	// roll anticlockwise to reach limit
	7:
		IF NOT(m_jointMounted[4]) THEN  
			// set target joint position
			m_targetMountPos[4]:=curJntPos[4]+m_mountMotionAng;
			// check if reach limit 
			IF i_slaveArm.filtJntCurrent[4]>m_maxJntCurrent THEN 
				m_jointMounted[4]:=TRUE;
				m_jntLimitPos3 := curJntPos[4];
				m_targetMountPos[4]:=curJntPos[4];
				m_jntOTG[4].init(m_targetMountPos[4], 0,m_instruMountVel, m_instruMountAcc, g_slaveArmCtrlCycleTime);
			END_IF
		END_IF
		IF NOT(m_jointMounted[5]) THEN 
			// set target joint position
			m_targetMountPos[5]:=curJntPos[5]-m_mountMotionAng;
			// check if reach limit 
			IF i_slaveArm.filtJntCurrent[5]<- m_maxJntCurrent THEN 
				m_jointMounted[5]:=TRUE;
				m_jntLimitPos4 := curJntPos[5];
				m_targetMountPos[5]:=curJntPos[5];
				m_jntOTG[5].init(m_targetMountPos[5], 0,m_instruMountVel, m_instruMountAcc, g_slaveArmCtrlCycleTime);
			END_IF	
		END_IF
		
		// transit
		IF m_jointMounted[4] AND m_jointMounted[5] THEN
			m_yawJntCaliStatus := 8;
			m_jointMounted[4]:=FALSE;
			m_jointMounted[5]:= FALSE;
		END_IF
		
	8:// calculate center/calibarted position
		m_targetMountPos[4] := (m_jntLimitPos1 + m_jntLimitPos3)/2-i_slaveArm.instrument.instruTypeInfo.m_instruYawBacklash/2.0;
		m_targetMountPos[5] := (m_jntLimitPos2 + m_jntLimitPos4)/2+i_slaveArm.instrument.instruTypeInfo.m_instruYawBacklash/2.0;
		m_yawJntCaliStatus := 9;

	9:
		IF ABS(m_targetMountPos[4]-curJntPos[4]) <GVL_SlaveControlParameters.g_jntCtrlAngTolLow  AND
			ABS(m_targetMountPos[5]-curJntPos[5]) <GVL_SlaveControlParameters.g_jntCtrlAngTolLow  THEN
			m_targetMountPos[4] := curJntPos[4]+i_slaveArm.instrument.instruTypeInfo.m_instruYawBacklash;
			m_yawJntCaliStatus := 19;
		END_IF
	19:
		IF ABS(m_targetMountPos[4]-curJntPos[4]) <GVL_SlaveControlParameters.g_jntCtrlAngTolLow  AND
			ABS(m_targetMountPos[5]-curJntPos[5]) <GVL_SlaveControlParameters.g_jntCtrlAngTolLow  THEN
			m_yawJntCaliStatus := 20;
		END_IF
	20: 
		m_targetMountPos[4] := curJntPos[4]+22.50*g_deg2Rad;
		m_targetMountPos[5] := curJntPos[5]+22.50*g_deg2Rad;
		IF ABS(m_targetMountPos[4]-m_cmdJntPos[4]) <GVL_SlaveControlParameters.g_jntCtrlAngTolLow  AND
			ABS(m_targetMountPos[5]-m_cmdJntPos[5]) <GVL_SlaveControlParameters.g_jntCtrlAngTolLow  THEN
			m_targetMountPos[4]:=curJntPos[4];
			m_targetMountPos[5]:=curJntPos[5];
			m_jntOTG[1].init(m_targetMountPos[4], 0,m_instruMountVel, m_instruMountAcc, g_slaveArmCtrlCycleTime);
			m_jntOTG[2].init(m_targetMountPos[5], 0,m_instruMountVel, m_instruMountAcc, g_slaveArmCtrlCycleTime);
		m_yawJntCaliStatus := 21;
 		END_IF
	21:
		m_targetMountPos[4] := curJntPos[4]-0.35*i_slaveArm.instrument.instruTypeInfo.m_maxGripAngle-i_slaveArm.instrument.instruTypeInfo.m_instruYawBacklash-25*g_deg2Rad;
		m_targetMountPos[5] := curJntPos[5]-0.35*i_slaveArm.instrument.instruTypeInfo.m_maxGripAngle-i_slaveArm.instrument.instruTypeInfo.m_instruYawBacklash-25*g_deg2Rad;
		m_yawJntCaliStatus := 22;
    22:
		IF ABS(m_targetMountPos[4]-m_cmdJntPos[4]) <GVL_SlaveControlParameters.g_jntCtrlAngTolLow  AND
			ABS(m_targetMountPos[5]-m_cmdJntPos[5]) <GVL_SlaveControlParameters.g_jntCtrlAngTolLow  THEN
		m_yawJntCaliStatus := 23;
 		END_IF
	23:// calculate center/calibarted position
		m_targetMountPos[4] := (m_jntLimitPos1 + m_jntLimitPos3)/2-i_slaveArm.instrument.instruTypeInfo.m_instruYawBacklash/2.0;
		m_targetMountPos[5] := (m_jntLimitPos2 + m_jntLimitPos4)/2+i_slaveArm.instrument.instruTypeInfo.m_instruYawBacklash/2.0;
		m_yawJntCaliStatus := 24;

	24:
		IF ABS(m_targetMountPos[4]-curJntPos[4]) <GVL_SlaveControlParameters.g_jntCtrlAngTolLow  AND
			ABS(m_targetMountPos[5]-curJntPos[5]) <GVL_SlaveControlParameters.g_jntCtrlAngTolLow  THEN
			m_targetMountPos[4] := curJntPos[4]+i_slaveArm.instrument.instruTypeInfo.m_instruYawBacklash;
			m_yawJntCaliStatus := 25;
		END_IF
	25:
		IF ABS(m_targetMountPos[4]-curJntPos[4]) <GVL_SlaveControlParameters.g_jntCtrlAngTolLow  AND
			ABS(m_targetMountPos[5]-curJntPos[5]) <GVL_SlaveControlParameters.g_jntCtrlAngTolLow  THEN
			m_yawJntCaliStatus := 10;
		END_IF
		
	// close finger	
	10:
			m_targetMountPos[4] := curJntPos[4]+gripCloseAng;
			m_targetMountPos[5] := curJntPos[5]+gripCloseAng;
			m_yawJntCaliStatus := 11;
	11:
		IF ABS(m_targetMountPos[4]-curJntPos[4]) <GVL_SlaveControlParameters.g_jntCtrlAngTolLow  AND
			ABS(m_targetMountPos[5]-curJntPos[5]) <GVL_SlaveControlParameters.g_jntCtrlAngTolLow  THEN
			m_yawJntCaliStatus := -1;
		END_IF

END_CASE

// traj plan
m_jntOTG[4].run(m_targetMountPos[4],0.0, o_cmdAcc=>m_cmdJntAcc[4],o_cmdVel=>m_cmdJntVel[4],o_cmdPos=>m_cmdJntPos[4]);
m_jntOTG[5].run(m_targetMountPos[5],0.0, o_cmdAcc=>m_cmdJntAcc[5],o_cmdVel=>m_cmdJntVel[5],o_cmdPos=>m_cmdJntPos[5]);
END_METHOD

END_FUNCTION_BLOCK

// ---- FBs_SlaveControllers/FB_SlaveArmCtrlBase.TcPOU
// Slave Arm Base Controller, Hold at Current Posture
FUNCTION_BLOCK FB_SlaveArmCtrlBase IMPLEMENTS I_SlaveArmCtrl
VAR_INPUT
END_VAR
VAR_OUTPUT
END_VAR
VAR
	// flag if the controller has finished all its jobs
	m_isFinished:BOOL:=FALSE;
	
	// controller execute time period
	m_timePeriod :LREAL:=0;
	
	// flag to hold last commands
	m_holdLastCmds :BOOL := FALSE;
	
	// arm control data
	// NOTE: simulated joint position is usd for kinematic controller 
	//		while command joint position is used for real robot controller
	// 		They are identical for the most time, but in some cases, simulated position is filted to get command one 
	m_simJntPos :Vec8d; 
	m_cmdJntPos : VEC8d; 
	m_cmdJntVel : VEC8d;
	m_cmdJntAcc : VEC8d;
	m_cmdJntTrq : VEC8d;
	m_jntOPMode : Vec8i;
	m_jntEnableFlag :Vec8i;
	m_cmdCartPose : ST_Frame;
	m_cmdCartTwist : Vec6d;
	m_FFJntTrq :Vec8d;
	
END_VAR

// override this function in each exact controller
METHOD PROTECTED calcCmdJntPos : BOOL
VAR_IN_OUT CONSTANT
	// endoscope pose in cart coordinate
	i_endoscopePose : ST_Frame;
	
	// master arm data
	i_masterStatus :ST_MasterStatus;
	
	// setup arm data
	i_setupStatus: ST_SetupStatus;
	
	// slave arm data
	i_slaveArm :FB_SlaveArm;
END_VAR
IF isFinished THEN
	RETURN;
END_IF
END_METHOD

// override this function in each exact controller
METHOD PROTECTED calcCmdJntTrq : BOOL
VAR_IN_OUT CONSTANT
	// endoscope pose in cart coordinate
	i_endoscopePose : ST_Frame;
	
	// master arm data
	i_masterStatus :ST_MasterStatus;
	
	// setup arm data
	i_setupStatus: ST_SetupStatus;
	
	// slave arm data
	i_slaveArm :FB_SlaveArm;
END_VAR
IF isFinished THEN
	RETURN;
END_IF

// set joint torque to zero in default
m_cmdJntTrq := g_zeroVec8d;
END_METHOD

METHOD checkToHoldLastCmds : BOOL
VAR_IN_OUT CONSTANT
	i_slaveArm :FB_SlaveArm;
END_VAR
VAR
	j:INT;
	maxJntErr:LREAL;
	jntCtrlErr:Vec8d;
END_VAR
// check if to hold the command joint position unchanged
vecSub(i_slaveArm.m_cmdJntPos, i_slaveArm.m_curJntPos,jntCtrlErr);
maxJntErr:=0.0;
FOR j:=1 TO g_sJntNum DO
	maxJntErr:= MAX(maxJntErr, ABS(jntCtrlErr[j]));
END_FOR

checkToHoldLastCmds := (maxJntErr<GVL_SlaveControlParameters.g_jntCtrlErrForCmdHold);
END_METHOD

METHOD copyCmds : BOOL
VAR_IN_OUT 
	r_slaveArmCtrlCmd :ST_SlaveArmCtrlCmds;
END_VAR
r_slaveArmCtrlCmd.m_jntEnableFlag :=m_jntEnableFlag;
r_slaveArmCtrlCmd.m_cmdCartPose:=m_cmdCartPose;
r_slaveArmCtrlCmd.m_cmdCartTwist:=m_cmdCartTwist;
r_slaveArmCtrlCmd.m_simJntPos:=m_simJntPos;
r_slaveArmCtrlCmd.m_cmdJntPos:=m_cmdJntPos;
r_slaveArmCtrlCmd.m_cmdJntVel:=m_cmdJntVel;
r_slaveArmCtrlCmd.m_cmdJntAcc:=m_cmdJntAcc;
r_slaveArmCtrlCmd.m_cmdJntTrq:=m_cmdJntTrq;
r_slaveArmCtrlCmd.m_jntOPMode:=m_jntOPMode;
r_slaveArmCtrlCmd.m_FFJntTrq:=m_FFJntTrq;
END_METHOD

// call this function to add friction compensation to m_cmdJntTrq
METHOD enableFrictionCompensation : BOOL
VAR_IN_OUT CONSTANT
	i_slaveArm :FB_SlaveArm;
END_VAR

VAR
	i:INT;
	frictionScale :LREAL;
END_VAR
// add joint friction compensation
FOR i:=1 TO g_sJntNum DO
	frictionScale :=LIMIT(-1.0, i_slaveArm.curJntVel[i]/g_fullFrictionVel,1.0);
	m_cmdJntTrq[i]:=m_cmdJntTrq[i]+frictionScale * g_frictionCompScale * GVL_SlaveArmDynamics.g_slaveJntFriction[i_slaveArm.armIdx, i];
END_FOR
END_METHOD

// override this function in each exact controller
// NOTICE: set joint control mode here, and do some initialization if needed
METHOD PUBLIC init : BOOL
VAR_IN_OUT CONSTANT
	i_slaveArm	:FB_SlaveArm;
END_VAR
VAR_IN_OUT 
	r_slaveArmCtrlCmd :ST_SlaveArmCtrlCmds;
END_VAR
m_timePeriod:=0;
m_jntEnableFlag :=g_onesVec8i;
m_jntEnableFlag[1] := 0;
m_jntEnableFlag[2] := 0;
m_jntEnableFlag[3] := 0;
m_jntOPMode:=g_slaveAllPosMode;
m_cmdCartPose:=i_slaveArm.curCartPose;
m_cmdCartTwist:=g_zeroVec6d;
IF FALSE = m_holdLastCmds THEN
	m_cmdJntPos:=i_slaveArm.curJntPos;
ELSE
	m_cmdJntPos:=r_slaveArmCtrlCmd.m_cmdJntPos;
END_IF
m_simJntPos := m_cmdJntPos;
m_cmdJntVel:=g_zeroVec8d;
m_cmdJntAcc:=g_zeroVec8d;
m_cmdJntTrq:=g_zeroVec8d;
m_FFJntTrq :=g_zeroVec8d;

// update commands to arm
copyCmds(r_slaveArmCtrlCmd);
END_METHOD

PROPERTY isFinished : BOOL
GET
isFinished:=m_isFinished;
END_GET
END_PROPERTY

{warning '添加方法实现'}
METHOD reset : BOOL
m_isFinished:=FALSE;
m_timePeriod:=0;
END_METHOD

{warning '添加方法实现'}
METHOD run : BOOL
VAR_IN_OUT CONSTANT
	i_endoscopePose : ST_Frame;
	i_masterStatus :ST_MasterStatus;
	i_setupStatus: ST_SetupStatus;
	i_slaveArm :FB_SlaveArm;
END_VAR
VAR_IN_OUT
	r_slaveArmCtrlCmd :ST_SlaveArmCtrlCmds;
END_VAR
VAR
	i:INT;
END_VAR
IF m_isFinished THEN
	RETURN;
END_IF

// check if arm enabled
IF FALSE = i_slaveArm.isEnabled(m_jntEnableFlag) THEN
	RETURN;
END_IF

// calculate command joint position--Motion control
calcCmdJntPos(i_endoscopePose, i_masterStatus, i_setupStatus, i_slaveArm);

// calculate command joint torque -- Force control
calcCmdJntTrq(i_endoscopePose, i_masterStatus, i_setupStatus, i_slaveArm);

// update commands to arm
copyCmds(r_slaveArmCtrlCmd);

// update time period
m_timePeriod := m_timePeriod+g_slaveArmCtrlCycleTime;
END_METHOD

PROPERTY timePeriod : Lreal
GET
timePeriod := m_timePeriod;
END_GET
END_PROPERTY

END_FUNCTION_BLOCK

// ---- FBs_SlaveControllers/FB_SlaveCtrlInstruEndoscopeTest.TcPOU
// Brief: Slave Arm test
FUNCTION_BLOCK PUBLIC FB_SlaveCtrlInstruEndoscopeTest EXTENDS FB_SlaveArmCtrlBase
VAR
																
	// final target DH joint position and grip angle
	m_targetDHJntPos:Vec3d;
	m_targetGripAng:LREAL;
	m_targetGripForceLevel :LREAL :=0;
	m_maxGripCurrent:LREAL:=350.0;
	m_maxGripCtrlCurrent:LREAL:=540.0;
	
	// interploated command joint position and grip angle 
	m_cmdDHJntPos :Vec6d;
	m_cmdDHJntVel :Vec6d;
	m_cmdGripAng:LREAL;

	// last joint position 
	m_lastCmdJntPos :Vec8d ;
	
	// instrument controller
	m_instruController : FB_BasicInstruControl;
	m_usKnifeController : FB_UltrosonicKnifeControl;
	m_instruCmdJntPos,m_instruCmdJntVel : Vec5d;
	m_instruCmdJntTrq :Vec5d;
	
	// OTG
	m_DHJntOTG:ARRAY[1..3] OF FB_secOrdTrajFilter;
	m_gripAngleOTG : FB_secOrdTrajFilter;
	m_maxJntVel:Vec3d:=[3(2.0)];
	m_maxJntAcc:Vec3d:=[3(4.0)];
	
	// instrument tyep
	m_instruType : E_InstrumentType;

	
	m_endoscopeAdjustment:BOOL;
	m_endoscopeOverturn:BOOL;
	m_endoscopeAdjustmentLast:BOOL;
	m_endoscopeOverturnLast:BOOL;
	
	m_tonEndoscopeOverturn:TON;
	m_endoscopeOverturn30:BOOL;
	m_endoscopeOverturn30Last:BOOL;
END_VAR

METHOD PROTECTED calcCmdJntPos : BOOL
VAR_IN_OUT CONSTANT
	i_endoscopePose : ST_Frame;
	i_masterStatus :ST_MasterStatus;
	i_setupStatus: ST_SetupStatus;
	i_slaveArm :FB_SlaveArm;
END_VAR

VAR 
	i:INT :=0;

END_VAR
//0/30°调整信号
IF (i_slaveArm.m_panelInstrumentOnIO  = 111) THEN      
	m_endoscopeAdjustment:=TRUE;
ELSE
	m_endoscopeAdjustment:=FALSE;
END_IF
//内窥镜翻转调整信号
IF (i_slaveArm.m_panelInstrumentOnIO =95) THEN    
	m_endoscopeOverturn:=TRUE;
ELSE
	m_endoscopeOverturn:=FALSE;
END_IF
m_tonEndoscopeOverturn(IN:=i_slaveArm.m_panelInstrumentOnIO  = 111,PT:=T#3S);
IF m_tonEndoscopeOverturn.Q THEN
	m_endoscopeOverturn30:=TRUE;
ELSE
	m_endoscopeOverturn30:=FALSE;
END_IF
//0/30°镜切换
IF m_endoscopeAdjustment AND NOT m_endoscopeAdjustmentLast THEN
	IF GVL_InstruTestUIVars.g_endoscopeAngle=0 THEN
		GVL_InstruTestUIVars.g_endoscopeAngle:=30;
	ELSE
		GVL_InstruTestUIVars.g_endoscopeAngle:=0;
	END_IF
END_IF
IF m_endoscopeOverturn30 AND NOT m_endoscopeOverturn30Last THEN
	IF GVL_InstruTestUIVars.g_endoscopeUpturn30FlagBit THEN
		m_targetDHJntPos[1]:=i_slaveArm.curDHJntPos[4]+30*g_deg2rad;
		GVL_InstruTestUIVars.g_endoscopeUpturn30FlagBit:=0;
	ELSE
		m_targetDHJntPos[1]:=i_slaveArm.curDHJntPos[4]-30*g_deg2rad;	
		GVL_InstruTestUIVars.g_endoscopeUpturn30FlagBit:=1;
	END_IF
END_IF
//内窥镜翻转信号
IF m_endoscopeOverturn AND NOT m_endoscopeOverturnLast THEN
	IF GVL_InstruTestUIVars.g_endoscopeUpturnFlagBit THEN
		m_targetDHJntPos[1]:=i_slaveArm.curDHJntPos[4]+180*g_deg2rad;
		GVL_InstruTestUIVars.g_endoscopeUpturnFlagBit:=0;
	ELSE
		m_targetDHJntPos[1]:=i_slaveArm.curDHJntPos[4]-180*g_deg2rad;	
		GVL_InstruTestUIVars.g_endoscopeUpturnFlagBit:=1;
	END_IF
END_IF
IF GVL_InstruTestUIVars.g_startEndoscopeTest THEN 
	m_targetDHJntPos[1]:=i_slaveArm.curDHJntPos[4]+GVL_InstruTestUIVars.g_cycleEndoscopeTest*2*pi;
	GVL_InstruTestUIVars.g_startEndoscopeTest:=0;
END_IF
m_endoscopeOverturnLast:=m_endoscopeOverturn;
m_endoscopeAdjustmentLast:=m_endoscopeAdjustment;
m_endoscopeOverturn30Last:=m_endoscopeOverturn30;
// run OTG
FOR i:=1 TO 3  DO
	m_DHJntOTG[i].run(m_targetDHJntPos[i],0.0, o_cmdAcc=>,o_cmdVel=>m_cmdDHJntVel[i],o_cmdPos=> m_cmdDHJntPos[i+3]);
END_FOR
m_gripAngleOTG.run(m_targetGripAng,0.0, o_cmdAcc=>,o_cmdVel=>,o_cmdPos=>m_cmdGripAng);
// calculate target motor joint position from DH joint position
i_slaveArm.instrument.instruIK(m_cmdDHJntPos,m_cmdGripAng, o_jntPos=>m_cmdJntPos);

// command velocity
vecSub(m_cmdJntPos, m_lastCmdJntPos, m_cmdJntVel);
vecSelfMultiNum(m_cmdJntVel, g_slaveArmCtrlFreq);
m_lastCmdJntPos:=m_cmdJntPos;
END_METHOD

// override this function in each exact controller
METHOD PROTECTED calcCmdJntTrq : BOOL
VAR_IN_OUT CONSTANT
	i_endoscopePose : ST_Frame;
	i_masterStatus :ST_MasterStatus;
	i_setupStatus: ST_SetupStatus;
	i_slaveArm :FB_SlaveArm;
END_VAR

VAR 
	nullspaceMat :Mat7d;
	ctrlTrq : Vec7d;
	i : int ;
END_VAR
// set joint torque to zero in default
m_cmdJntTrq := g_zeroVec8d;

// instrument joint control
FOR i:=1 TO 5 DO 
	m_instruCmdJntPos[i]:=m_cmdJntPos[i+3];
	m_instruCmdJntVel[i]:=m_cmdJntVel[i+3];
END_FOR

IF i_slaveArm.instrument.instruType = InstruType_UltrasoundKnifeS OR i_slaveArm.instrument.instruType = InstruType_UltrasoundKnifeU THEN
	m_usKnifeController.run(m_instruCmdJntPos,m_instruCmdJntVel, m_targetGripForceLevel, i_slaveArm, o_cmdJntTrq=>m_instruCmdJntTrq);
ELSE
	m_instruController.run(m_instruCmdJntPos,m_instruCmdJntVel, m_cmdDHJntPos[6], m_cmdDHJntVel[6], m_targetGripForceLevel, i_slaveArm, o_cmdJntTrq=>m_instruCmdJntTrq);
END_IF

FOR i:=1 TO 5 DO
	m_cmdJntTrq[i+3]:=m_instruCmdJntTrq[i];
	m_cmdJntTrq[6]:=0;
END_FOR
END_METHOD

METHOD PUBLIC init : BOOL
VAR_IN_OUT CONSTANT
	i_slaveArm	:FB_SlaveArm;
END_VAR
VAR_IN_OUT 
	r_slaveArmCtrlCmd :ST_SlaveArmCtrlCmds;
END_VAR

VAR
	i:int;
END_VAR
SUPER^.Init(i_slaveArm,r_slaveArmCtrlCmd);
m_lastCmdJntPos:=m_cmdJntPos;
m_jntOPMode[1] := DriverOPMode_PosTrq;
m_jntOPMode[2] := DriverOPMode_PosTrq;
m_jntOPMode[3] := DriverOPMode_PosTrq;
m_jntOPMode[4] := DriverOPMode_Trq;
m_jntOPMode[5] := DriverOPMode_Trq;
m_jntOPMode[6] := DriverOPMode_Trq;
m_jntOPMode[7] := DriverOPMode_Trq;
m_jntOPMode[8] := DriverOPMode_Trq;

m_cmdDHJntPos :=i_slaveArm.curDHJntPos;
m_cmdDHJntVel :=g_zeroVec6d;
m_targetGripAng := i_slaveArm.curGripAngle;
m_targetDHJntPos[1] := i_slaveArm.curDHJntPos[4];
m_targetDHJntPos[2] := i_slaveArm.curDHJntPos[5];
m_targetDHJntPos[3] := i_slaveArm.curDHJntPos[6];

// init instrument controller
m_instruController.init(i_slaveArm,m_maxGripCurrent,m_maxGripCtrlCurrent);
m_usKnifeController.init(i_slaveArm);

FOR i:=1 TO 3  DO
	m_DHJntOTG[i].init(m_cmdDHJntPos[i+3], 0, m_maxJntVel[i], m_maxJntAcc[i], g_slaveArmCtrlCycleTime);
END_FOR

m_gripAngleOTG.init(m_targetGripAng, 0, 2*m_maxJntVel[3], 2*m_maxJntAcc[3], g_slaveArmCtrlCycleTime);
// update commands to arm
copyCmds(r_slaveArmCtrlCmd);
END_METHOD

PROPERTY InstruBacklash : Vec5d
GET
IF m_instruType = InstruType_UltrasoundKnifeS OR m_instruType = InstruType_UltrasoundKnifeU THEN
	instruBacklash := g_zeroVec5d;
ELSE
	instruBacklash := m_instruController.m_jntBacklash;
END_IF
END_GET
END_PROPERTY

END_FUNCTION_BLOCK

// ---- FBs_SlaveControllers/FB_SlaveCtrlInstruManualTest.TcPOU
// Brief: Slave Arm test
FUNCTION_BLOCK PUBLIC FB_SlaveCtrlInstruManualTest EXTENDS FB_SlaveArmCtrlBase
VAR
																
	// final target DH joint position and grip angle
	m_targetDHJntPos:Vec3d;
	m_targetGripAng:LREAL;
	m_targetGripForceLevel :LREAL :=0;
	
	// interploated command joint position and grip angle 
	m_cmdDHJntPos :Vec6d;
	m_cmdDHJntVel :Vec6d;
	m_cmdGripAng:LREAL;

	// last joint position 
	m_lastCmdJntPos :Vec8d ;
	
	// instrument controller
	m_instruController : FB_BasicInstruControl;
	m_usKnifeController : FB_UltrosonicKnifeControl;
	m_instruCmdJntPos,m_instruCmdJntVel : Vec5d;
	m_instruCmdJntTrq :Vec5d;
	
	// OTG
	m_DHJntOTG:ARRAY[1..3] OF FB_secOrdTrajFilter;
	m_gripAngleOTG : FB_secOrdTrajFilter;
	m_maxJntVel:Vec3d:=[3(2.0)];
	m_maxJntAcc:Vec3d:=[3(4.0)];
	
	// instrument tyep
	m_instruType : E_InstrumentType;
	bStart: BOOL;
	iStep: INT;
	fbTon: TON;

	m_maxGripCurrent:LREAL:=350.0;
	m_maxGripCtrlCurrent:LREAL:=540.0;
END_VAR

METHOD PROTECTED calcCmdJntPos : BOOL
VAR_IN_OUT CONSTANT
	i_endoscopePose : ST_Frame;
	i_masterStatus :ST_MasterStatus;
	i_setupStatus: ST_SetupStatus;
	i_slaveArm :FB_SlaveArm;
END_VAR

VAR 
	i:INT :=0;
	errThres :LREAL;
	m_targetDHJntPosLast: Vec3d;
	m_curCmdDHJntPos: Vec3d;
	m_compensationAngleDH: Vec3d;
	m_targetGripAngLast: LREAL;
	m_curCmdAng: LREAL;

END_VAR
// determine target DH joint position and gripper motion
IF GVL_InstruTestUIVars.g_moveToSetPosFlag THEN
	m_targetDHJntPos[1] := GVL_InstruTestUIVars.g_targetRollAng*g_deg2rad;
	m_targetDHJntPos[2] := (GVL_InstruTestUIVars.g_targetPitchAng-90)*g_deg2rad;
	m_targetDHJntPos[3] := GVL_InstruTestUIVars.g_targetYawAng*g_deg2rad;
	IF GVL_InstruTestUIVars.g_targetGripAng>-15 AND GVL_InstruTestUIVars.g_targetGripAng<100  THEN 
		m_targetGripAng := GVL_InstruTestUIVars.g_targetGripAng*g_deg2rad;
		m_targetGripForceLevel:=0;
	ELSIF GVL_InstruTestUIVars.g_targetGripAng<=-15 AND GVL_InstruTestUIVars.g_targetGripAng>=-100 THEN 
		m_targetGripAng := -15*g_deg2rad;
		m_targetGripForceLevel := LIMIT(0, ABS(GVL_InstruTestUIVars.g_targetGripAng), 100);
	ELSIF GVL_InstruTestUIVars.g_targetGripAng<-101 THEN 
		m_targetGripAng := 60 *g_deg2rad;
		m_targetGripForceLevel := LIMIT(-100, 100+GVL_InstruTestUIVars.g_targetGripAng, 0);
	END_IF
ELSIF GVL_InstruTestUIVars.g_gripperOpenFlag THEN
	m_targetGripAng := i_slaveArm.instrument.instruTypeInfo.m_maxGripAngle;
	m_targetGripForceLevel :=0;
ELSIF GVL_InstruTestUIVars.g_gripperCloseFlag THEN
	m_targetGripAng := 0;
	m_targetGripForceLevel :=0;
ELSIF GVL_InstruTestUIVars.g_maxGripForceFlag THEN
	m_targetGripAng := -45*g_deg2rad;
	m_targetGripForceLevel :=100;
END_IF

IF GVL_InstruTestUIVars.m_cycleStart THEN 
	bStart:=TRUE;
	GVL_InstruTestUIVars.m_cycleStart:=FALSE;
END_IF
IF GVL_InstruTestUIVars.m_cycleStop THEN 
	bStart:=FALSE;
	GVL_InstruTestUIVars.m_cycleStop:=FALSE;
END_IF
fbTon(IN:=iStep=10,PT:=T#1S);
IF bStart THEN
	CASE iStep OF 
		0:
			m_targetGripAng := i_slaveArm.instrument.instruTypeInfo.m_maxGripAngle;
			m_targetGripForceLevel :=0;
			iStep:=5;
		5:
		    IF ABS(m_cmdGripAng- m_targetGripAng)< g_jntCtrlAngTolLow THEN
				iStep:=10;
			END_IF
		10:
			IF fbTon.Q THEN
				m_targetGripAng := -90*g_deg2rad;
				m_targetGripForceLevel :=0;
				iStep:=15;
			END_IF
		15:
		    IF ABS(m_cmdGripAng- m_targetGripAng)< g_jntCtrlAngTolLow THEN
				iStep:=0;
			END_IF
	END_CASE
END_IF
// run OTG
FOR i:=1 TO 3  DO
	m_DHJntOTG[i].run(m_targetDHJntPos[i],0.0, o_cmdAcc=>,o_cmdVel=>m_cmdDHJntVel[i],o_cmdPos=> m_cmdDHJntPos[i+3]);
END_FOR
m_gripAngleOTG.run(m_targetGripAng,0.0, o_cmdAcc=>,o_cmdVel=>,o_cmdPos=>m_cmdGripAng);

// calculate target motor joint position from DH joint position
i_slaveArm.instrument.instruIK(m_cmdDHJntPos,m_cmdGripAng, o_jntPos=>m_cmdJntPos);

// command velocity
vecSub(m_cmdJntPos, m_lastCmdJntPos, m_cmdJntVel);
vecSelfMultiNum(m_cmdJntVel, g_slaveArmCtrlFreq);
m_lastCmdJntPos:=m_cmdJntPos;
END_METHOD

// override this function in each exact controller
METHOD PROTECTED calcCmdJntTrq : BOOL
VAR_IN_OUT CONSTANT
	i_endoscopePose : ST_Frame;
	i_masterStatus :ST_MasterStatus;
	i_setupStatus: ST_SetupStatus;
	i_slaveArm :FB_SlaveArm;
END_VAR

VAR 
	nullspaceMat :Mat7d;
	ctrlTrq : Vec7d;
	i : int ;
END_VAR
// set joint torque to zero in default
m_cmdJntTrq := g_zeroVec8d;

// instrument joint control
FOR i:=1 TO 5 DO 
	m_instruCmdJntPos[i]:=m_cmdJntPos[i+3];
	m_instruCmdJntVel[i]:=m_cmdJntVel[i+3];
END_FOR

IF i_slaveArm.instrument.instruType = InstruType_UltrasoundKnifeS OR i_slaveArm.instrument.instruType = InstruType_UltrasoundKnifeU THEN
	m_usKnifeController.run(m_instruCmdJntPos,m_instruCmdJntVel, m_targetGripForceLevel, i_slaveArm, o_cmdJntTrq=>m_instruCmdJntTrq);
ELSE
	m_instruController.run(m_instruCmdJntPos,m_instruCmdJntVel, m_cmdDHJntPos[6], m_cmdDHJntVel[6], m_targetGripForceLevel, i_slaveArm, o_cmdJntTrq=>m_instruCmdJntTrq);
END_IF

FOR i:=1 TO 5 DO
	m_cmdJntTrq[i+3]:=m_instruCmdJntTrq[i];
END_FOR
END_METHOD

METHOD PUBLIC init : BOOL
VAR_IN_OUT CONSTANT
	i_slaveArm	:FB_SlaveArm;
END_VAR
VAR_IN_OUT 
	r_slaveArmCtrlCmd :ST_SlaveArmCtrlCmds;
END_VAR

VAR
	i:int;
END_VAR
SUPER^.Init(i_slaveArm,r_slaveArmCtrlCmd);
m_lastCmdJntPos:=m_cmdJntPos;
m_jntOPMode[1] := DriverOPMode_PosTrq;
m_jntOPMode[2] := DriverOPMode_PosTrq;
m_jntOPMode[3] := DriverOPMode_PosTrq;
m_jntOPMode[4] := DriverOPMode_Trq;
m_jntOPMode[5] := DriverOPMode_Trq;
m_jntOPMode[6] := DriverOPMode_Trq;
m_jntOPMode[7] := DriverOPMode_Trq;
m_jntOPMode[8] := DriverOPMode_Trq;

m_cmdDHJntPos :=i_slaveArm.curDHJntPos;
m_cmdDHJntVel :=g_zeroVec6d;
m_targetGripAng := i_slaveArm.curGripAngle;
m_targetDHJntPos[1] := i_slaveArm.curDHJntPos[4];
m_targetDHJntPos[2] := i_slaveArm.curDHJntPos[5];
m_targetDHJntPos[3] := i_slaveArm.curDHJntPos[6];

// init instrument controller
m_instruController.init(i_slaveArm,m_maxGripCurrent,m_maxGripCtrlCurrent);
m_usKnifeController.init(i_slaveArm);
iStep:=0;
bStart:=FALSE;
IF GVL_InstruTestUIVars.g_rotationAngularVel=0 THEN GVL_InstruTestUIVars.g_rotationAngularVel:=5;END_IF
IF GVL_InstruTestUIVars.g_pitchAngularVel=0 THEN GVL_InstruTestUIVars.g_pitchAngularVel:=5;END_IF
IF GVL_InstruTestUIVars.g_deviationAngularVel=0 THEN GVL_InstruTestUIVars.g_deviationAngularVel:=5;END_IF
IF GVL_InstruTestUIVars.g_rotationAngularAcc=0 THEN GVL_InstruTestUIVars.g_rotationAngularAcc:=30;END_IF
IF GVL_InstruTestUIVars.g_pitchAngularAcc=0 THEN GVL_InstruTestUIVars.g_pitchAngularAcc:=30;END_IF
IF GVL_InstruTestUIVars.g_deviationAngularAcc=0 THEN GVL_InstruTestUIVars.g_deviationAngularAcc:=30;END_IF
FOR i:=1 TO 3  DO
	m_maxJntVel[i]:=5;
	m_maxJntAcc[i]:=30;
	IF GVL_InstruTestUIVars.g_account.actualPermission=2 THEN
		m_maxJntVel[1]:=GVL_InstruTestUIVars.g_rotationAngularVel;
		m_maxJntVel[2]:=GVL_InstruTestUIVars.g_pitchAngularVel;
		m_maxJntVel[3]:=GVL_InstruTestUIVars.g_deviationAngularVel;
		m_maxJntAcc[1]:=GVL_InstruTestUIVars.g_rotationAngularAcc;
		m_maxJntAcc[2]:=GVL_InstruTestUIVars.g_pitchAngularAcc;
		m_maxJntAcc[3]:=GVL_InstruTestUIVars.g_deviationAngularAcc;
	END_IF
END_FOR

FOR i:=1 TO 3  DO
	m_DHJntOTG[i].init(m_cmdDHJntPos[i+3], 0, m_maxJntVel[i], m_maxJntAcc[i], g_slaveArmCtrlCycleTime);
END_FOR

m_gripAngleOTG.init(m_targetGripAng, 0, 2*m_maxJntVel[3], 2*m_maxJntAcc[3], g_slaveArmCtrlCycleTime);
// update commands to arm
copyCmds(r_slaveArmCtrlCmd);
END_METHOD

PROPERTY InstruBacklash : Vec5d
GET
IF m_instruType = InstruType_UltrasoundKnifeS OR m_instruType = InstruType_UltrasoundKnifeU THEN
	instruBacklash := g_zeroVec5d;
ELSE
	instruBacklash := m_instruController.m_jntBacklash;
END_IF
END_GET
END_PROPERTY

END_FUNCTION_BLOCK

// ---- FBs_SlaveControllers/FB_SlaveCtrlMountInstru.TcPOU
// Brief: Mounting Instrument
FUNCTION_BLOCK PUBLIC FB_SlaveCtrlMountInstru EXTENDS FB_SlaveArmCtrlBase
VAR
	// mount status
	m_instruMountStatus :INT := 0;
	m_scopeMountStatus :INT := 0;
	m_ultrasoundMountStatus :INT :=0 ;
	
	// flag if joint is mounted
	m_jointMounted :ARRAY[1..5] OF BOOL := [5(FALSE)];
	
	// instrument mount motion range
	m_mountMotionAng :Vec5d :=[5(pi)];
	
	// instrument mount direction
	m_mountDir :Vec5i :=[1, 1, 1, 1, 1];
	
	// mount motion planning
	m_jntOTG :ARRAY[1..5] OF FB_secOrdTrajFilter;
	m_instruMountVel :LREAL := 4*PI;
	m_instruMountAcc :LREAL := 8*PI;
	
	//Joint 4 half-range angle of instrument
	m_instruJnt4HalfRangeAng :LREAL := 323*g_deg2Rad;
	
	// joint current threshold which indicate panel is buckled with instrument
	m_maxJntCurrent :Vec5d := [220, 220, 120, 120, 120];
	m_maxJntCurrentOldEndoScope :Vec5d := [200, 200, 200, 350, 350];
	
	// command mount motion
	m_targetMountPos :Vec8d;
	
	// instrument zero position
	m_instruZeroDeviation :Vec5d;
	
	//ultrasound knife Reduce the current rotation Angle  J3
	m_ultraKnifeRotaAngleJ3 :LREAL := 30*g_deg2Rad;
	
	// ultrasound knife rotate angle zero position
	m_ultraKnifeRotAngZeroPos :LREAL := 4.50567;
	
	// joint position error
	m_jntPosErr :Vec5d;
	m_linkSingleErr:Vec5d;
	
	// endoscope motion angle to original position
	m_scopeJnt4CenterMotionAng :LREAL :=175*g_deg2Rad;
	m_scopeJnt5CenterMotionAng :LREAL :=150*g_deg2Rad;
	
	//instrument clamp error Id
	m_instruClampErrId : UINT;
	m_instruClampTime : LREAL;
	m_noCurrentTime : LREAL :=5;
	m_notReturnToZero : LREAL :=10;
	m_maxClampTime :LREAL :=0.5;
	m_endoscopeClampDelay :Vec5d;
END_VAR

// override this function in each exact controller
METHOD PROTECTED calcCmdJntPos : BOOL
VAR_IN_OUT CONSTANT
	i_endoscopePose : ST_Frame;
	i_masterStatus :ST_MasterStatus;
	i_setupStatus: ST_SetupStatus;
	i_slaveArm :FB_SlaveArm;
END_VAR

VAR 
END_VAR
// mount error detect;
m_instruClampErrId := instruClampStatus(i_slaveArm);

// return directly if instrument/endoscope is not readed
IF NOT(i_slaveArm.instrument.onChipData.m_InstruReadSucceed) THEN
	return;
END_IF

IF i_slaveArm.instrument.onChipData.m_InstruReadSucceed AND InstruType_endoscope = i_slaveArm.instrument.onChipData.m_InstruID THEN
	mountEndoscope(i_slaveArm);
ELSIF i_slaveArm.instrument.onChipData.m_InstruReadSucceed AND InstruType_NewEndoscope = i_slaveArm.instrument.onChipData.m_InstruID THEN
	mountNewEndoscope(i_slaveArm);
ELSIF i_slaveArm.instrument.onChipData.m_InstruReadSucceed AND (InstruType_UltrasoundKnifeS = i_slaveArm.instrument.m_instruType OR InstruType_UltrasoundKnifeU = i_slaveArm.instrument.m_instruType) THEN
	mountUltraKnife(i_slaveArm);
ELSE
	mountInstrument(i_slaveArm);
END_IF
END_METHOD

// override this function in each exact controller
METHOD PROTECTED calcCmdJntTrq : BOOL
VAR_IN_OUT CONSTANT
	i_endoscopePose : ST_Frame;
	i_masterStatus :ST_MasterStatus;
	i_setupStatus: ST_SetupStatus;
	i_slaveArm :FB_SlaveArm;
END_VAR
VAR
	i :INT;
END_VAR
// set joint torque to zero in default
m_cmdJntTrq := g_zeroVec8d;

// clear instrument joint torque if  mount fail
IF m_instruClampErrId >0 THEN 
	FOR i:=4 TO 8 DO 
		m_jntOPMode[i] := DriverOPMode_Trq;
		m_cmdJntPos[i] := i_slaveArm.curJntPos[i];
		m_cmdJntTrq[i]:= i_slaveArm.curJntTrq[i]*0.8;
	END_FOR
	m_instruClampTime := m_instruClampTime + g_slaveArmCtrlCycleTime;
	m_isFinished := m_instruClampTime > m_maxClampTime;
END_IF
END_METHOD

METHOD PUBLIC init : BOOL
VAR_IN_OUT CONSTANT
	i_slaveArm	:FB_SlaveArm;
END_VAR
VAR_IN_OUT 
	r_slaveArmCtrlCmd :ST_SlaveArmCtrlCmds;
END_VAR

VAR
	i : INT;
END_VAR
// check if to hold the command joint position unchanged
m_holdLastCmds := checkToHoldLastCmds(i_slaveArm);

SUPER^.Init(i_slaveArm,r_slaveArmCtrlCmd);
m_jntOPMode[4] := DriverOPMode_PosTrq;
m_jntOPMode[5] := DriverOPMode_PosTrq;
m_jntOPMode[6] := DriverOPMode_PosTrq;
m_jntOPMode[7] := DriverOPMode_PosTrq;
m_jntOPMode[8] := DriverOPMode_PosTrq;

FOR i:=1 TO 5 DO
	m_targetMountPos[i+3]:=m_cmdJntPos[i+3];
	m_jntOTG[i].init(m_targetMountPos[i+3], 0,m_instruMountVel, m_instruMountAcc, g_slaveArmCtrlCycleTime);
	m_jointMounted[i]:=FALSE;
	m_endoscopeClampDelay[i] := 0;
END_FOR

m_instruMountStatus:=0;
m_scopeMountStatus:=0;
m_ultrasoundMountStatus:=0;
m_instruClampErrId := 0;
m_instruClampTime := 0;
// update commands to arm
copyCmds(r_slaveArmCtrlCmd);

//other 
GVL_InstruTestUIVars.g_endoscopeAngle:=0;
GVL_InstruTestUIVars.g_endoscopeUpturnFlagBit:=FALSE;
GVL_InstruTestUIVars.g_endoscopeUpturn30FlagBit:=FALSE;
END_METHOD

PROPERTY instruClampErrId :  UINT
GET
instruClampErrId := m_instruClampErrId;
END_GET
SET
m_instruClampErrId:=instruClampErrId;
END_SET
END_PROPERTY

METHOD instruClampStatus : UINT
VAR_IN_OUT CONSTANT
	i_slaveArm :FB_SlaveArm;
END_VAR
//m_instruClampErrId=1 instrumen clamp the current does not reach the set value
//m_instruClampErrId=2 instrumen clamp position does not return to zero
//m_instruClampErrId=3 instrumen can not be recongnized

IF i_slaveArm.instrument.onChipData.m_InstruReadSucceed THEN
	IF InstruType_endoscope = i_slaveArm.instrument.m_instruType THEN
		IF (m_scopeMountStatus=0 OR m_scopeMountStatus=1) AND m_timePeriod>=m_noCurrentTime  THEN
			instruClampStatus := 1;
		ELSIF m_scopeMountStatus=3 AND m_timePeriod>=m_notReturnToZero  THEN
			instruClampStatus := 2;
		END_IF
		
	ELSIF (InstruType_UltrasoundKnifeS = i_slaveArm.instrument.m_instruType OR InstruType_UltrasoundKnifeU = i_slaveArm.instrument.m_instruType) THEN
		IF (m_ultrasoundMountStatus=0) AND m_timePeriod>=m_noCurrentTime  THEN
			instruClampStatus := 1;
		ELSIF (m_scopeMountStatus=3) AND m_timePeriod>=m_notReturnToZero  THEN
			instruClampStatus := 2;
		END_IF
			
	ELSE
		IF (m_instruMountStatus=0) AND m_timePeriod>=m_noCurrentTime  THEN
			instruClampStatus := 1;
		ELSIF (m_instruMountStatus=3) AND m_timePeriod>=m_notReturnToZero  THEN
			instruClampStatus := 2;
		END_IF
	END_IF

ELSIF i_slaveArm.instrument.onChipData.m_Error = TRUE THEN
	instruClampStatus:=3;
END_IF
END_METHOD

METHOD mountEndoscope : BOOL
VAR_IN_OUT CONSTANT
	i_slaveArm :FB_SlaveArm;
END_VAR

VAR 
	i :INT;
	curJntPos :Vec8d;
END_VAR
curJntPos := i_slaveArm.curJntPos;

CASE m_scopeMountStatus OF
	//fix scope lock joint(joint 7)
	0:
		// other joints stay still
		FOR i:=1 TO 3 DO
			m_jointMounted[i] := TRUE;
			m_targetMountPos[i+3]:=curJntPos[i+3];
			m_jntOTG[i].init(m_targetMountPos[i+3], 0,m_instruMountVel, m_instruMountAcc, g_slaveArmCtrlCycleTime);
		END_FOR
	
		// check if buckled
		m_jointMounted[4]:=FALSE; 
		m_jointMounted[5]:=FALSE; 
		IF ABS(i_slaveArm.filtJntCurrent[7])> m_maxJntCurrentOldEndoScope[4] THEN 
			m_jointMounted[4]:=TRUE;
			m_targetMountPos[7]:=curJntPos[7];
			m_jntOTG[4].init(m_targetMountPos[7], 0,m_instruMountVel, m_instruMountAcc, g_slaveArmCtrlCycleTime);
			m_scopeMountStatus:=1;
		ELSE
			m_targetMountPos[7]:=curJntPos[7]+m_mountMotionAng[4];
		END_IF

	1: // buckle scope rotate joint (joint 8)
		m_jointMounted[5]:=FALSE; 
		IF ABS(i_slaveArm.filtJntCurrent[8])> m_maxJntCurrentOldEndoScope[5] THEN 
			m_jointMounted[5]:=TRUE;
			m_targetMountPos[8]:=curJntPos[8];
			m_jntOTG[5].init(m_targetMountPos[8], 0,m_instruMountVel, m_instruMountAcc, g_slaveArmCtrlCycleTime);
			m_scopeMountStatus:=2;
		ELSE
			m_targetMountPos[8]:=curJntPos[8]+m_mountMotionAng[5];
		END_IF
	

	2:// move back to zero position
		m_targetMountPos[7]:= curJntPos[7]-m_scopeJnt4CenterMotionAng;
		m_targetMountPos[8]:= curJntPos[8]-m_scopeJnt5CenterMotionAng;
		m_scopeMountStatus :=3;
		
		
	3:
		IF ABS(m_targetMountPos[7]-curJntPos[7]) <GVL_SlaveControlParameters.g_jntCtrlAngTolHigh AND 
				ABS(m_targetMountPos[8]-curJntPos[8]) <GVL_SlaveControlParameters.g_jntCtrlAngTolHigh THEN
			// record current joint position as offset for instrument
			i_slaveArm.instrument.initInstruJntPos(i_slaveArm.curJntPos);
			m_isFinished := TRUE;
		END_IF
		
END_CASE

// traj plan
FOR i:=1 TO 5 DO
	m_jntOTG[i].run(m_targetMountPos[i+3],0.0, o_cmdAcc=>m_cmdJntAcc[3+i],o_cmdVel=>m_cmdJntVel[3+i],o_cmdPos=>m_cmdJntPos[i+3]);
END_FOR
END_METHOD

METHOD mountInstrument : BOOL
VAR_IN_OUT CONSTANT
	i_slaveArm :FB_SlaveArm;
END_VAR

VAR 
	i :INT;
	curJntPos :Vec8d;
END_VAR
curJntPos := i_slaveArm.curJntPos;

// joint4 stay still if instrument has only on finger
IF i_slaveArm.instrument.instruTypeInfo.m_isSingleFinger THEN
	m_jointMounted[1]:=TRUE;
END_IF

CASE m_instruMountStatus OF
	// To lock panel with instrument
	0:
		//buckle panel with instrument
		FOR i:=1 TO 5 DO
			// check if buckled 
			IF (i= 4 AND ABS(i_slaveArm.filtJntCurrent[i+3])> m_maxJntCurrent[i] AND ABS(i_slaveArm.curJntVel[i+3])<1.0*g_deg2Rad) 
				OR (i<> 4 AND ABS(i_slaveArm.filtJntCurrent[i+3])> m_maxJntCurrent[i] )THEN 
				m_jointMounted[i]:=TRUE;
			END_IF
			
			// set target joint position
			IF FALSE = m_jointMounted[i] THEN
					m_targetMountPos[i+3]:=curJntPos[i+3]-m_mountMotionAng[i];	
			ELSE
					m_targetMountPos[i+3]:=curJntPos[i+3];
					m_jntOTG[i].init(m_targetMountPos[i+3], 0,m_instruMountVel, m_instruMountAcc, g_slaveArmCtrlCycleTime);
			END_IF
		END_FOR
		
		
		// check transition condition
		IF (m_jointMounted[1] AND m_jointMounted[2] AND m_jointMounted[3] AND m_jointMounted[4] AND m_jointMounted[5])  THEN
			IF i_slaveArm.instrument.onChipData.m_InstruReadSucceed THEN//Check whether the data is read successfully
				IF i_slaveArm.instrument.instruTypeInfo.m_isSingleFinger THEN
					m_instruMountStatus:=1;
				ELSE
					m_instruMountStatus:=20;
				END_IF
			END_IF
		END_IF

	20: 
		m_targetMountPos[4] := curJntPos[4]+22.5*g_deg2Rad;
		m_targetMountPos[5] := curJntPos[5]+22.5*g_deg2Rad;
		IF ABS(m_targetMountPos[4]-m_cmdJntPos[4]) <GVL_SlaveControlParameters.g_jntCtrlAngTolLow  AND
			ABS(m_targetMountPos[5]-m_cmdJntPos[5]) <GVL_SlaveControlParameters.g_jntCtrlAngTolLow  THEN
			m_targetMountPos[4]:=curJntPos[4];
			m_targetMountPos[5]:=curJntPos[5];
			m_jntOTG[1].init(m_targetMountPos[4], 0,m_instruMountVel, m_instruMountAcc, g_slaveArmCtrlCycleTime);
			m_jntOTG[2].init(m_targetMountPos[5], 0,m_instruMountVel, m_instruMountAcc, g_slaveArmCtrlCycleTime);
			m_instruMountStatus := 21;
 		END_IF
	21:
		m_targetMountPos[4] := curJntPos[4]-0.35*i_slaveArm.instrument.instruTypeInfo.m_maxGripAngle-i_slaveArm.instrument.instruTypeInfo.m_instruYawBacklash-35*g_deg2Rad;
		m_targetMountPos[5] := curJntPos[5]-0.35*i_slaveArm.instrument.instruTypeInfo.m_maxGripAngle-i_slaveArm.instrument.instruTypeInfo.m_instruYawBacklash-35*g_deg2Rad;
		m_instruMountStatus := 22;
    22:
		IF ABS(m_targetMountPos[4]-m_cmdJntPos[4]) <GVL_SlaveControlParameters.g_jntCtrlAngTolLow  AND
			ABS(m_targetMountPos[5]-m_cmdJntPos[5]) <GVL_SlaveControlParameters.g_jntCtrlAngTolLow  THEN
		m_instruMountStatus := 1;
 		END_IF
		
	1:// calculation deviates from the instrument zero position
		FOR i:=1 TO 5 DO
			m_instruZeroDeviation[i] :=  i_slaveArm.linkSingle[i+3] - i_slaveArm.instrument.onChipData.m_InstruPos[i];
		END_FOR
		m_instruMountStatus :=2;
	
	2:// move back to zero position
		FOR i:=1 TO 3 DO//J1-3
			IF m_instruZeroDeviation[i]>pi THEN
				m_instruZeroDeviation[i] := m_instruZeroDeviation[i] - 2*PI;
			ELSIF m_instruZeroDeviation[i]<-pi THEN
				m_instruZeroDeviation[i] := m_instruZeroDeviation[i] + 2*PI;
			END_IF
		END_FOR
		
		//joint4
		IF m_instruZeroDeviation[4]>0 AND m_instruZeroDeviation[4] < pi THEN
			m_instruZeroDeviation[4] := m_instruZeroDeviation[4] - 2*pi;
		ELSIF m_instruZeroDeviation[4]<0 AND m_instruZeroDeviation[4] > -pi THEN
			m_instruZeroDeviation[4] := m_instruZeroDeviation[4] + 2*pi;
		END_IF
		
		FOR i:=1 TO 5 DO
			m_targetMountPos[i+3]:=curJntPos[i+3] - m_instruZeroDeviation[i];
		END_FOR
		m_instruMountStatus :=3;
		
	3: // move to zero position
		m_instruMountStatus :=4;
		FOR i:=1 TO 4 DO 
			m_jntPosErr[i]:=m_targetMountPos[i+3]-curJntPos[i+3];
			m_linkSingleErr[i] := ABS( i_slaveArm.linkSingle[i+3] - i_slaveArm.instrument.onChipData.m_InstruPos[i]);
			m_linkSingleErr[i]:= MIN(m_linkSingleErr[i], g_2pi-m_linkSingleErr[i]);
			IF ABS(m_jntPosErr[i]) >5*GVL_SlaveControlParameters.g_jntCtrlAngTolLow OR 	ABS( m_linkSingleErr[i]) >5*g_deg2rad THEN
				m_instruMountStatus :=3;
				EXIT;
			END_IF
		END_FOR
	
	4:
		// record current joint position as offset for instrument
		i_slaveArm.instrument.initInstruJntPos(i_slaveArm.curJntPos);
		
		m_isFinished :=  TRUE;

END_CASE

// traj plan
FOR i:=1 TO 5 DO
	m_jntOTG[i].run(m_targetMountPos[i+3],0.0, o_cmdAcc=>m_cmdJntAcc[3+i],o_cmdVel=>m_cmdJntVel[3+i],o_cmdPos=>m_cmdJntPos[i+3]);
END_FOR
END_METHOD

METHOD mountNewEndoscope : BOOL
VAR_IN_OUT CONSTANT
	i_slaveArm :FB_SlaveArm;
END_VAR

VAR 
	i :INT;
	curJntPos :Vec8d;
END_VAR
curJntPos := i_slaveArm.curJntPos;

CASE m_scopeMountStatus OF
	//fix scope lock joint(joint 7)
	0:
		// other joints stay still
		FOR i:=1 TO 5 DO
			IF i = 1 OR i =2 OR i =5 THEN
				m_jointMounted[i] := TRUE;
				m_targetMountPos[i+3]:=curJntPos[i+3];
				m_jntOTG[i].init(m_targetMountPos[i+3], 0,m_instruMountVel, m_instruMountAcc, g_slaveArmCtrlCycleTime);
			END_IF
		END_FOR
	
		// check if buckled
		FOR i:=3 TO 4 DO
			IF ABS(i_slaveArm.filtJntCurrent[i+3])> m_maxJntCurrent[i] THEN 
				m_endoscopeClampDelay[i] := m_endoscopeClampDelay[i] + g_slaveArmCtrlCycleTime;
				IF m_endoscopeClampDelay[i] > 0.5 THEN
					m_jointMounted[i]:=TRUE;
					m_targetMountPos[i+3]:=curJntPos[i+3];
					m_jntOTG[i].init(m_targetMountPos[i+3], 0,m_instruMountVel, m_instruMountAcc, g_slaveArmCtrlCycleTime);
				END_IF
			ELSE
				m_targetMountPos[i+3]:=curJntPos[i+3]+m_mountMotionAng[i]/5;
			END_IF
		END_FOR
		
		IF m_jointMounted[3] AND m_jointMounted[4] THEN
			m_targetMountPos[6]:=curJntPos[6]-0.1;
			m_targetMountPos[7]:=curJntPos[7]-0.1;
			m_scopeMountStatus:=4;
		END_IF
	4:
		
		m_endoscopeClampDelay[1] := m_endoscopeClampDelay[1] + g_slaveArmCtrlCycleTime;
		IF m_endoscopeClampDelay[1] > 0.5 THEN
			m_jntOPMode[7] := DriverOPMode_PosTrq;
			m_scopeMountStatus:=1;
		END_IF

	1: // buckle scope rotate joint (joint 8)
		m_jntOPMode[6] := DriverOPMode_Trq;
		IF i_slaveArm.instrument.onChipData.m_InstruPos[1] <> 0 THEN
			m_instruZeroDeviation[4] :=  i_slaveArm.linkSingle[7] - i_slaveArm.instrument.onChipData.m_InstruPos[1];
		ELSE
			m_instruZeroDeviation[4] :=  i_slaveArm.linkSingle[7] - i_slaveArm.instrument.onChipData.m_InstruPos[4]+0.1;
		END_IF
		
		m_scopeMountStatus :=2;

	2:// move back to zero position
		
		//joint4
		IF m_instruZeroDeviation[4]>0 AND m_instruZeroDeviation[4] > pi THEN
			m_instruZeroDeviation[4] := m_instruZeroDeviation[4] - 2*pi;
		ELSIF m_instruZeroDeviation[4]<0 AND m_instruZeroDeviation[4] < -pi THEN
			m_instruZeroDeviation[4] := m_instruZeroDeviation[4] + 2*pi;
		END_IF
		
		m_targetMountPos[7]:=curJntPos[7] - m_instruZeroDeviation[4];
		m_scopeMountStatus :=3;
		
		
	3:
		m_isFinished := FALSE;
		IF ABS(m_targetMountPos[7]-curJntPos[7]) <GVL_SlaveControlParameters.g_jntCtrlAngTolHigh/10 THEN
			// record current joint position as offset for instrument
			i_slaveArm.instrument.initInstruJntPos(i_slaveArm.curJntPos);
			m_scopeMountStatus :=4;
			m_isFinished := TRUE;
		END_IF
		
END_CASE

// traj plan
FOR i:=1 TO 5 DO
	m_jntOTG[i].run(m_targetMountPos[i+3],0.0, o_cmdAcc=>m_cmdJntAcc[3+i],o_cmdVel=>m_cmdJntVel[3+i],o_cmdPos=>m_cmdJntPos[i+3]);
END_FOR

IF m_jntOPMode[6] = DriverOPMode_Trq THEN
	m_cmdJntTrq[6] := -i_slaveArm.cmdJntTrq[7];
END_IF
END_METHOD

METHOD mountUltraKnife : BOOL
VAR_IN_OUT CONSTANT
	i_slaveArm :FB_SlaveArm;
END_VAR

VAR 
	i :INT;
	curJntPos :Vec8d;
END_VAR
curJntPos := i_slaveArm.curJntPos;

m_jointMounted[1]:=TRUE;
m_jointMounted[2]:=TRUE;


CASE m_ultrasoundMountStatus OF 
	// To lock panel with instrument
	0:
		//buckle panel with instrument
		FOR i:=3 TO 5 DO
			// check if buckled 
			IF ABS(i_slaveArm.filtJntCurrent[i+3])> m_maxJntCurrent[i] THEN 
				m_jointMounted[i]:=TRUE;
				m_targetMountPos[i+3]:=curJntPos[i+3];
				m_jntOTG[i].init(m_targetMountPos[i+3], 0,m_instruMountVel, m_instruMountAcc, g_slaveArmCtrlCycleTime);
			END_IF
			
			// set target joint position
			IF FALSE = m_jointMounted[i] THEN
				IF i = 5 THEN
					m_targetMountPos[i+3]:=curJntPos[i+3]+m_mountMotionAng[i];
				ELSE
					m_targetMountPos[i+3]:=curJntPos[i+3]-m_mountMotionAng[i];
				END_IF
				
			END_IF
		END_FOR

		// check transition condition
		IF ( m_jointMounted[3] AND m_jointMounted[4] AND m_jointMounted[5] )  THEN
			IF i_slaveArm.instrument.onChipData.m_InstruReadSucceed THEN//Check whether the data is read successfully
				m_ultrasoundMountStatus:=1;
			END_IF
		END_IF

	1:
		//m_jntOPMode[8] := DriverOPMode_Trq;
		// calculation deviates from the instrument zero position
		m_instruZeroDeviation[3] :=  i_slaveArm.linkSingle[6] - i_slaveArm.instrument.onChipData.m_InstruPos[3]; //m_ultraKnifeRotaAngleJ3;
		m_instruZeroDeviation[4] :=  i_slaveArm.linkSingle[7] - m_ultraKnifeRotAngZeroPos;
		m_ultrasoundMountStatus :=2;
		
	2:// move back to zero position
		//joint3
		IF m_instruZeroDeviation[3] > 2*pi THEN
			m_instruZeroDeviation[3] := m_instruZeroDeviation[3] - 2*pi  ;
		ELSIF  m_instruZeroDeviation[3] < -pi THEN
			m_instruZeroDeviation[3] := 2*pi + m_instruZeroDeviation[3] ;
		END_IF
		//joint4
		IF m_instruZeroDeviation[4]>0 AND m_instruZeroDeviation[4] < pi THEN
			m_instruZeroDeviation[4] := m_instruZeroDeviation[4] - 2*pi;
		ELSIF m_instruZeroDeviation[4]<0 AND m_instruZeroDeviation[4] > -pi THEN
			m_instruZeroDeviation[4] := m_instruZeroDeviation[4] + 2*pi;
		END_IF
	
		// set target joint position
		m_targetMountPos[6]:=curJntPos[6] - m_instruZeroDeviation[3];
		//m_targetMountPos[6]:=curJntPos[6] + m_ultraKnifeRotaAngleJ3;
		m_targetMountPos[7]:=curJntPos[7] - m_instruZeroDeviation[4];
		m_targetMountPos[8]:=curJntPos[8] - m_instruZeroDeviation[4];

		m_ultrasoundMountStatus :=3;

	3:
		// joint8 in passive mode
		m_jntOPMode[8] := DriverOPMode_Trq;
		
		m_isFinished:=TRUE;
		FOR i:=3 TO 4 DO 
			m_jntPosErr[i]:=m_targetMountPos[i+3]-curJntPos[i+3];
			IF ABS(m_jntPosErr[i]) >GVL_SlaveControlParameters.g_jntCtrlAngTolLow  THEN
				m_isFinished := FALSE;
				EXIT;
			END_IF
		END_FOR	
		
		// record current joint position as offset for instrument
		i_slaveArm.instrument.initInstruJntPos(i_slaveArm.curJntPos);

END_CASE


// traj plan
FOR i:=1 TO 5 DO
	m_jntOTG[i].run(m_targetMountPos[i+3],0.0, o_cmdAcc=>m_cmdJntAcc[3+i],o_cmdVel=>m_cmdJntVel[3+i],o_cmdPos=>m_cmdJntPos[i+3]);
END_FOR
END_METHOD

END_FUNCTION_BLOCK

// ---- FBs_SlaveControllers/FB_SlaveCtrlPowerBoxCalibration.TcPOU
// Brief: Mounting Panel
FUNCTION_BLOCK PUBLIC FB_SlaveCtrlPowerBoxCalibration EXTENDS FB_SlaveArmCtrlBase
VAR_INPUT
END_VAR
VAR_OUTPUT
END_VAR
VAR
	// powerBoxCalibration status
	m_powerBoxCalibrationStatus :INT := 0;
	
	// flag if joint is mounted
	m_jointMounted :ARRAY[1..5] OF BOOL := [5(FALSE)];
	
	// mount motion planning
	m_jntOTG :ARRAY[1..5] OF FB_secOrdTrajFilter;
	m_panelMountVel :LREAL := 2*pi;
	m_panelMountAcc :LREAL := 4*pi;
	
	// joint current threshold which indicate motor is buckled with panel
	m_maxJntCurrent :INT := 220;
	
	// command mount motion
	m_powerBoxCalibrationStepPos :LREAL := 45.0 * g_deg2Rad;
	m_targetPowerBoxCalibrationPos :Vec5d;
END_VAR

// override this function in each exact controller
METHOD PROTECTED calcCmdJntPos : BOOL
VAR_IN_OUT CONSTANT
	i_endoscopePose : ST_Frame;
	i_masterStatus :ST_MasterStatus;
	i_setupStatus: ST_SetupStatus;
	i_slaveArm :FB_SlaveArm;
END_VAR

VAR 
	i :INT;
	curJntPos :Vec8d;
END_VAR

curJntPos := i_slaveArm.curJntPos;

CASE m_powerBoxCalibrationStatus OF
	// To lock joint with panel
	0:
		FOR i:=1 TO 5 DO
			// check joint buckled with panel
			IF ABS(i_slaveArm.filtJntCurrent[i+3])> m_maxJntCurrent THEN 
				m_jointMounted[i]:=TRUE;
				m_targetPowerBoxCalibrationPos[i]:=curJntPos[i+3];
				m_jntOTG[i].init(m_targetPowerBoxCalibrationPos[i], 0,m_panelMountVel, m_panelMountAcc, g_slaveArmCtrlCycleTime);
			END_IF
			
			// set command joint position step
			IF FALSE = m_jointMounted[i] THEN
				m_targetPowerBoxCalibrationPos[i]:=curJntPos[i+3]+m_powerBoxCalibrationStepPos;
			END_IF
		END_FOR
		
		IF m_jointMounted[1]AND m_jointMounted[2]AND m_jointMounted[3] AND m_jointMounted[4] AND m_jointMounted[5]THEN
			m_powerBoxCalibrationStatus:=1;
		END_IF
	1:
		m_isFinished:=TRUE;
END_CASE

// traj plan
FOR i:=1 TO 5 DO
	m_jntOTG[i].run(m_targetPowerBoxCalibrationPos[i],0.0, o_cmdAcc=>m_cmdJntAcc[3+i],o_cmdVel=>m_cmdJntVel[3+i],o_cmdPos=>m_cmdJntPos[i+3]);
END_FOR
END_METHOD

METHOD PUBLIC init : BOOL
VAR_IN_OUT CONSTANT
	i_slaveArm	:FB_SlaveArm;
END_VAR
VAR_IN_OUT 
	r_slaveArmCtrlCmd :ST_SlaveArmCtrlCmds;
END_VAR
VAR
	i : INT;
END_VAR
SUPER^.Init(i_slaveArm,r_slaveArmCtrlCmd);//T
m_jntOPMode[4] := DriverOPMode_PosTrq;
m_jntOPMode[5] := DriverOPMode_PosTrq;
m_jntOPMode[6] := DriverOPMode_PosTrq;
m_jntOPMode[7] := DriverOPMode_PosTrq;
m_jntOPMode[8] := DriverOPMode_PosTrq;

m_powerBoxCalibrationStatus:=0;
FOR i:=1 TO 5 DO
	m_targetPowerBoxCalibrationPos[i]:=m_cmdJntPos[i+3];
	m_jntOTG[i].init(m_targetPowerBoxCalibrationPos[i], 0,m_panelMountVel, m_panelMountAcc, g_slaveArmCtrlCycleTime);
	m_jointMounted[i]:=FALSE;
END_FOR

// update commands to arm
copyCmds(r_slaveArmCtrlCmd);
END_METHOD

END_FUNCTION_BLOCK

// ---- FBs_SlaveControllers/FB_SlaveCtrlStop.TcPOU
// Brief: Slave Arm Joint1-3 decelerate to stop
FUNCTION_BLOCK PUBLIC FB_SlaveCtrlStop EXTENDS FB_SlaveArmCtrlBase
VAR
	// stop motion is terminated after set time period
	m_maxStopPeriod :LREAL := 0.12;
	
	// deceleration period 
	m_decPeriod :LREAL := 0.1;
	
	// instrument joint compensated backlash
	m_instruBacklash :Vec5d :=g_zeroVec5d;

END_VAR

// override this function in each exact controller
METHOD PROTECTED calcCmdJntPos : BOOL
VAR_IN_OUT CONSTANT
	i_endoscopePose : ST_Frame;
	i_masterStatus :ST_MasterStatus;
	i_setupStatus: ST_SetupStatus;
	i_slaveArm :FB_SlaveArm;
END_VAR

VAR 
	i :INT;
	nextCmdVel :LREAL;
END_VAR
IF m_isFinished THEN
	m_cmdJntVel := g_zeroVec8d;
	m_cmdJntPos := i_slaveArm.curJntPos;
	m_FFJntTrq := g_zeroVec8d;
	RETURN;
END_IF

IF m_timePeriod > m_maxStopPeriod  THEN
	m_isFinished := TRUE;
	RETURN;
END_IF

FOR i := 1 TO 3 DO
	IF m_timePeriod > m_decPeriod THEN
		m_cmdJntVel[i] := 0;
		m_FFJntTrq[i]:=0;
	ELSE
		nextCmdVel := m_cmdJntVel[i] + m_cmdJntAcc[i]*g_slaveArmCtrlCycleTime;
		m_cmdJntPos[i] := m_cmdJntPos[i] + (nextCmdVel + m_cmdJntVel[i])*g_slaveArmCtrlCycleTime/2.0;
		m_cmdJntVel[i] := nextCmdVel;
		m_FFJntTrq[i] :=  i_slaveArm.massMat[i,i] * m_cmdJntAcc[i] ;
	END_IF
END_FOR
END_METHOD

METHOD PUBLIC init : BOOL
VAR_IN_OUT CONSTANT
	i_slaveArm	:FB_SlaveArm;
END_VAR
VAR_IN_OUT 
	r_slaveArmCtrlCmd :ST_SlaveArmCtrlCmds;
END_VAR
VAR
	i:INT;
	maxJntTrq:LREAL;
END_VAR
SUPER^.Init(i_slaveArm,r_slaveArmCtrlCmd);

// determine joint deceleration
FOR i:=1 TO 3 DO 
	m_jntOPMode[i] := DriverOPMode_PosTrq;
	m_cmdJntVel[i] := i_slaveArm.curJntVel[i];
	i_slaveArm.m_jntPIDCtrl[i].reset();
	m_cmdJntAcc[i] := -i_slaveArm.curJntVel[i]/m_decPeriod;
END_FOR

// NOTE: move instrument joint to remove backlash compensation
IF i_slaveArm.instrument.instruType = InstruType_Endoscope THEN
	m_instruBacklash := g_zeroVec5d;
ELSE
	FOR i:=4 TO 7 DO 
		m_jntOPMode[i] := DriverOPMode_PosTrq;
		m_cmdJntPos[i] := i_slaveArm.curJntPos[i]-m_instruBacklash[i-3];
	END_FOR
END_IF


// update commands to arm
copyCmds(r_slaveArmCtrlCmd);
END_METHOD

METHOD setInstruBacklash : BOOL
VAR_INPUT
	i_backlash :Vec5d;
END_VAR
m_instruBacklash := i_backlash;
END_METHOD

END_FUNCTION_BLOCK

// ---- FBs_SlaveControllers/FB_SlaveCtrlTest.TcPOU
// Brief: Slave Arm test
FUNCTION_BLOCK PUBLIC FB_SlaveCtrlTest EXTENDS FB_SlaveArmCtrlBase
VAR_INPUT
END_VAR
VAR_OUTPUT
END_VAR
VAR
// ################ variables for single DH  joint test ##################
	m_enableFrictionComp :BOOL :=false;
	m_freqTestFlag :BOOL:=FALSE;
	m_initJntPos :Vec6d;
	m_cmdDHJntPos :Vec6d;
	m_cmdDHJntVel :Vec6d;
	m_cmdGripAng:LREAL;
	m_jntMotionFreq :Vec6d :=[0.2, 0.2, 0.1, 3(0.1)];
	m_jntMotionRange :Vec6d :=[pi/6, pi/6, 0.1, 3(pi/6)];
	m_testJntIdx :INT :=1;
	m_gripperAngle : LREAL :=0;
	m_gripForceLevel :LREAL :=0;
	m_lastCmdJntPos :Vec8d ;
	
	m_stepTestFlag :BOOL :=FALSE;
	m_jntStep : LREAL := 5*g_deg2Rad;
	
	// instrument controller
	m_instruController : FB_BasicInstruControl;
	m_usKnifeController : FB_UltrosonicKnifeControl;
	m_instruCmdJntPos,m_instruCmdJntVel : Vec5d;
	m_instruCmdJntTrq :Vec5d;
	m_maxGripCurrent:LREAL:=350.0;
	m_maxGripCtrlCurrent:LREAL:=540.0;
	
	m_errCmdPos, m_errCurPos :LREAL;
	m_errPosIdx : INT;
	
	m_originalJntPos:Vec8d;
		m_jntOTG:array[1..6] of FB_secOrdTrajFilter;
		m_gripAngleOTG : FB_secOrdTrajFilter;
	
//####################################################################

END_VAR

METHOD PROTECTED calcCmdJntPos : BOOL
VAR_IN_OUT CONSTANT
	i_endoscopePose : ST_Frame;
	i_masterStatus :ST_MasterStatus;
	i_setupStatus: ST_SetupStatus;
	i_slaveArm :FB_SlaveArm;
END_VAR

VAR 
	i:INT :=0;
	errThres :LREAL;

END_VAR
IF m_testJntIdx <4 OR m_testJntIdx >6 THEN
	RETURN;
END_IF

// frequency test
IF m_freqTestFlag THEN 
	m_cmdDHJntPos[m_testJntIdx]:=m_initJntPos[m_testJntIdx]+m_jntMotionRange[m_testJntIdx]/2
									+0.5*m_jntMotionRange[m_testJntIdx]*SIN(2*pi*m_jntMotionFreq[m_testJntIdx]*m_timePeriod-pi/2);
	m_cmdDHJntVel[m_testJntIdx]:=0.5*m_jntMotionRange[m_testJntIdx]*2*pi*m_jntMotionFreq[m_testJntIdx]*COS(2*pi*m_jntMotionFreq[m_testJntIdx]*m_timePeriod-pi/2);
// step test
ELSIF m_stepTestFlag THEN;
	m_jntOTG[m_testJntIdx].run(m_initJntPos[m_testJntIdx]+m_jntStep,0.0, o_cmdAcc=>,o_cmdVel=>m_cmdDHJntVel[m_testJntIdx],o_cmdPos=> m_cmdDHJntPos[m_testJntIdx]);
// reset controller
ELSE
	m_timePeriod:=0;
	m_initJntPos :=i_slaveArm.curDHJntPos;
	m_originalJntPos := i_slaveArm.curJntPos;
	m_cmdDHJntPos :=m_initJntPos;
	m_cmdDHJntVel :=g_zeroVec6d;
	m_gripperAngle := i_slaveArm.curGripAngle;
	// init instrument controller
	m_instruController.init(i_slaveArm,m_maxGripCurrent,m_maxGripCtrlCurrent);
	m_usKnifeController.init(i_slaveArm);
	
	FOR i:=1 TO 6  DO
		m_jntOTG[i].init(m_initJntPos[i], 0,12, 100, g_slaveArmCtrlCycleTime);
	END_FOR
	
	m_gripAngleOTG.init(m_gripperAngle, 0, 2, 8, g_slaveArmCtrlCycleTime);
END_IF

// calculate target motor joint position from DH joint position
m_gripAngleOTG.run(m_gripperAngle,0.0, o_cmdAcc=>,o_cmdVel=>,o_cmdPos=>m_cmdGripAng);
i_slaveArm.instrument.instruIK(m_cmdDHJntPos,m_cmdGripAng, o_jntPos=>m_cmdJntPos);

// command velocity
vecSub(m_cmdJntPos, m_lastCmdJntPos, m_cmdJntVel);
vecSelfMultiNum(m_cmdJntVel, g_slaveArmCtrlFreq);
m_lastCmdJntPos:=m_cmdJntPos;
END_METHOD

// override this function in each exact controller
METHOD PROTECTED calcCmdJntTrq : BOOL
VAR_IN_OUT CONSTANT
	i_endoscopePose : ST_Frame;
	i_masterStatus :ST_MasterStatus;
	i_setupStatus: ST_SetupStatus;
	i_slaveArm :FB_SlaveArm;
END_VAR

VAR 
	nullspaceMat :Mat7d;
	ctrlTrq : Vec7d;
	i : int ;
END_VAR
// set joint torque to zero in default
m_cmdJntTrq := g_zeroVec8d;

// instrument joint control
FOR i:=1 TO 5 DO 
	m_instruCmdJntPos[i]:=m_cmdJntPos[i+3];
	m_instruCmdJntVel[i]:=m_cmdJntVel[i+3];
END_FOR

IF i_slaveArm.instrument.instruType = InstruType_UltrasoundKnifeS OR i_slaveArm.instrument.instruType = InstruType_UltrasoundKnifeU THEN
	m_usKnifeController.run(m_instruCmdJntPos,m_instruCmdJntVel, m_gripForceLevel, i_slaveArm, o_cmdJntTrq=>m_instruCmdJntTrq);
ELSE
	m_instruController.run(m_instruCmdJntPos,m_instruCmdJntVel, m_cmdDHJntPos[6], m_cmdDHJntVel[6], m_gripForceLevel, i_slaveArm, o_cmdJntTrq=>m_instruCmdJntTrq);
END_IF

FOR i:=1 TO 5 DO
	m_cmdJntTrq[i+3]:=m_instruCmdJntTrq[i];
END_FOR

// add friction
IF m_enableFrictionComp THEN
	enableFrictionCompensation(i_slaveArm);
END_IF
END_METHOD

METHOD PUBLIC init : BOOL
VAR_IN_OUT CONSTANT
	i_slaveArm	:FB_SlaveArm;
END_VAR
VAR_IN_OUT 
	r_slaveArmCtrlCmd :ST_SlaveArmCtrlCmds;
END_VAR

VAR
	i:int;
END_VAR
SUPER^.Init(i_slaveArm,r_slaveArmCtrlCmd);
m_lastCmdJntPos:=m_cmdJntPos;
m_jntOPMode[1] := DriverOPMode_PosTrq;
m_jntOPMode[2] := DriverOPMode_PosTrq;
m_jntOPMode[3] := DriverOPMode_PosTrq;
m_jntOPMode[4] := DriverOPMode_Trq;
m_jntOPMode[5] := DriverOPMode_Trq;
m_jntOPMode[6] := DriverOPMode_Trq;
m_jntOPMode[7] := DriverOPMode_Trq;
m_jntOPMode[8] := DriverOPMode_Trq;

m_initJntPos :=i_slaveArm.curDHJntPos;
m_originalJntPos := i_slaveArm.curJntPos;
m_cmdDHJntPos :=m_initJntPos;
m_cmdDHJntVel :=g_zeroVec6d;
m_gripperAngle := i_slaveArm.curGripAngle;

// init instrument controller
m_instruController.init(i_slaveArm,m_maxGripCurrent,m_maxGripCtrlCurrent);
m_usKnifeController.init(i_slaveArm);

FOR i:=1 TO 6  DO
	m_jntOTG[i].init(m_initJntPos[i], 0,12, 100, g_slaveArmCtrlCycleTime);
END_FOR

m_gripAngleOTG.init(m_gripperAngle, 0,2, 8, g_slaveArmCtrlCycleTime);
// update commands to arm
copyCmds(r_slaveArmCtrlCmd);
END_METHOD

END_FUNCTION_BLOCK

// ---- FBs_SlaveControllers/FB_SlaveCtrlError.TcPOU
// Brief: Slave Arm Error Hold
FUNCTION_BLOCK PUBLIC FB_SlaveCtrlError EXTENDS FB_SlaveArmCtrlBase
VAR
	// velocity for full damping
	m_maxAdjustVel :Vec3d := [1.2, 1.2, 0.3];
	
	// velocity start to enable damping
	m_velLBForDamp :Vec3d := [1.0, 1.0, 0.2];
	
	// max damp
	m_maxDamp :Vec3d := [50, 50, 500];
	
	// distance buffer from joint limit to start damp
	m_limitBufferForDamp :Vec3d :=[20*g_deg2Rad, 20*g_deg2Rad, 0.03];
END_VAR

// override this function in each exact controller
METHOD PROTECTED calcCmdJntPos : BOOL
VAR_IN_OUT CONSTANT
	// endoscope pose in cart coordinate
	i_endoscopePose : ST_Frame;
	
	// master arm data
	i_masterStatus :ST_MasterStatus;
	
	// setup arm data
	i_setupStatus: ST_SetupStatus;
	
	// slave arm data
	i_slaveArm :FB_SlaveArm;
END_VAR
VAR
	i:INT;
END_VAR
m_cmdJntPos := i_slaveArm.curJntPos;
END_METHOD

// override this function in each exact controller
METHOD PROTECTED calcCmdJntTrq : BOOL
VAR_IN_OUT CONSTANT
	i_endoscopePose : ST_Frame;
	i_masterStatus :ST_MasterStatus;
	i_setupStatus: ST_SetupStatus;
	i_slaveArm :FB_SlaveArm;
END_VAR
VAR
	i :INT;
	dampScale :LREAL;
	limitDis :LREAL;
END_VAR
// set joint torque to zero in default
m_cmdJntTrq := g_zeroVec8d;

// enable joint adjust if its error is recoverable
FOR i:=1 TO 3 DO
	// disable joint
	IF NOT(i_slaveArm.adjustOn) THEN
		m_jntEnableFlag[i]:= 0;
		m_jntOPMode[i]:=DriverOPMode_Pos;
		CONTINUE;
	END_IF
	
	// enable joint
	m_jntEnableFlag[i]:= 1;
	m_jntOPMode[i]:=DriverOPMode_Trq;
	
	// add damp near joint limit
	IF (i_slaveArm.curJntPos[i] > GVL_SlaveMotorParameters.g_maxDHJntPos[i] - m_limitBufferForDamp[i] AND  i_slaveArm.curJntVel[i]> 0 ) 
		OR (i_slaveArm.curJntPos[i] < GVL_SlaveMotorParameters.g_minDHJntPos[i] + m_limitBufferForDamp[i] AND  i_slaveArm.curJntVel[i]<0 )  THEN
		limitDis := MIN(GVL_SlaveMotorParameters.g_maxDHJntPos[i] - i_slaveArm.curJntPos[i], i_slaveArm.curJntPos[i]-GVL_SlaveMotorParameters.g_minDHJntPos[i]);
		dampScale  :=LIMIT(0, 1-limitDis/m_limitBufferForDamp[i],1);
		m_cmdJntTrq[i]:= -dampScale * m_maxDamp[i] * i_slaveArm.curJntVel[i];
	END_IF

	// compute damp
	IF ABS(i_slaveArm.curJntVel[i]) > m_velLBForDamp[i] THEN 
		dampScale:=LIMIT(0, (ABS(i_slaveArm.curJntVel[i])- m_velLBForDamp[i])/(m_maxAdjustVel[i] - m_velLBForDamp[i]), 1 );
		m_cmdJntTrq[i] :=m_cmdJntTrq[i] -i_slaveArm.curJntVel[i] * m_maxDamp[i] * dampScale;
	END_IF

END_FOR
END_METHOD

// override this function in each exact controller
// NOTICE: set joint control mode here, and do some initialization if needed
METHOD PUBLIC init : BOOL
VAR_IN_OUT CONSTANT
	i_slaveArm	:FB_SlaveArm;
END_VAR
VAR_IN_OUT 
	r_slaveArmCtrlCmd :ST_SlaveArmCtrlCmds;
END_VAR


VAR
	i:INT;
END_VAR
SUPER^.Init(i_slaveArm,r_slaveArmCtrlCmd);

// disable first three joints
m_jntEnableFlag[1]:= 0;
m_jntEnableFlag[2]:= 0;
m_jntEnableFlag[3]:= 0;

// disable instrument joints which is in error 
//FOR i:=4 TO g_sJntNum DO
//	IF SafetyCheck.m_SafetyCheck.m_jntErrFlag[i_slaveArm.armIdx, i+g_setupJntNum, 2] OR  SafetyCheck.m_SafetyCheck.m_jntErrFlag[i_slaveArm.armIdx, i+g_setupJntNum, 3] THEN
//		m_jntEnableFlag[i] := 0;
//	ELSE
//		m_jntEnableFlag[i] := 1;
//	END_IF
//END_FOR
 
 // update commands to arm
copyCmds(r_slaveArmCtrlCmd);
END_METHOD

END_FUNCTION_BLOCK

// ---- FBs_SlaveControllers/FB_SlaveCtrlMasterSlave.TcPOU
// Brief: Slave Arm MasterSlave controller
FUNCTION_BLOCK PUBLIC FB_SlaveCtrlMasterSlave EXTENDS FB_SlaveArmCtrlBase
VAR_INPUT
END_VAR
VAR_OUTPUT
END_VAR
VAR
	// minimum distance between instrument tip and remote center
	m_minInstruRCDis:LREAL := 0.05;
	
	// master-slave motion scale
	m_MSMotionScale :LREAL;
		
	// gripper match angle threshold
	m_gripperMatchAngThres :LREAL := 2*g_deg2Rad;
	
	// control error thershold from joint limit back to free space
	m_jntLimitOriErr :LREAL :=g_deg2Rad * 5;
	
	// master-slave error thershold to halt control 
	m_safetyOriErr :LREAL :=g_deg2Rad * 150;
	
	// filter cut-off frequency for master-slave control
	m_macroCmdJntPosLpfCutoffFreq : LREAL :=5;
	m_microCmdJntPosLpfCutoffFreq : LREAL :=15;
	
	// last command joint position
	m_lastCmdJntPos :Vec8d;
	
	// simulated DH joint position
	m_simDHJntPos : Vec6d;
	
	// simulated slave twist of DH joint
	m_simDHJointVel :Vec6d;
		
	// enter master-slave control for the first time
	m_firstIn :BOOL := TRUE;
	
	// flag if reach joint limit
	m_reachMacroJntLimit :BOOL;
	m_reachWristJntLimit :BOOL;
	
	// master/slave origin pose when first enter master-slave control
	m_masterOriginPose : ST_Frame;
	m_slaveOriginPose : ST_Frame;
	
	// orientation deviation(in master coordinate) between master and slave when first enter control
	m_MSOriDeviation : Mat3d;
	
	// command joint position filter
	m_cmdJntPosLpf:ARRAY[1..8] OF FB_LowPassFilter;
	
	// commmand yaw angle and velocity
	m_cmdYawAngle :LREAL;
	m_cmdYawVel :LREAL;
	
	// comand yaw angle and velocity filter
	m_cmdYawAngLpf : FB_LowPassFilter;
	m_cmdYawVelLpf : FB_LowPassFilter;
	
	// master pose/velocity in monitor coordinate
	m_masterPose :ST_Frame;
	m_masterTwist : Vec6d;
	
	// master grip angle
	m_masterGripAngle : LREAL;
	
	// slave command/current pose in endoscope coordinate
	m_slaveCmdPoseInScope :ST_Frame;
	m_slavePoseInScope : ST_Frame;
	
	// slave command/current pose in cart
	m_slaveCmdPoseInCart :ST_Frame;
	m_slavePoseInCart : ST_Frame;
	
	// instrument controller
	m_basicInstruController : FB_BasicInstruControl;
	m_usKnifeController : FB_UltrosonicKnifeControl;
	
	// slave command grip angle and grip force level
	m_slaveCmdGripAngle :LREAL;
	m_slaveCmdGripForceLevel:LREAL;
	
	// slave pose error
	m_slavePosErr :Vec3d;
	m_slaveRotErr :Mat3d;
	m_errAngle : LREAL;
	m_errAxisLocal, m_errAxis :Vec3d;
	m_masterSlavePoseError :Vec6d;
	
	// velocity for slave to track master motion
	m_slaveTrackTwist :Vec6d;
	m_slaveCmdVel, m_slaveCmdWVel : Vec3d;
	
	// flag to start gripper control
	m_gripperCtrlFlag :BOOL;
	
	//################# variable to interpolate master pose ##############
	m_firstInterpolate :BOOL :=TRUE;
	m_lastMasterPose : ST_Frame;
	m_lastMasterGripAngle :LREAL;
	m_masterInterpolateCycle :INT := 4;
	m_curInterpolateCylce :INT := 1;
	m_masterPosInterStep :Vec3d;
	m_masterOriInterStep :Mat3d;
	m_masterGripAngleInterStep :LREAL;
	m_interplotedMasterPose :ST_Frame;
	m_interplotedMasterGripAngle :LREAL;
	
	
	// code execute time measure
	m_codeTime : Profiler;
	
END_VAR

END_FUNCTION_BLOCK

// ---- FBs_SlaveControllers/FB_SlaveCtrlAdjust.TcPOU
// Brief: Slave Arm Adjust
FUNCTION_BLOCK PUBLIC FB_SlaveCtrlAdjust EXTENDS FB_SlaveArmCtrlBase
VAR
	// velocity for full damping
	m_maxAdjustVel :Vec3d := [1.2, 1.2, 0.3];
	
	// velocity start to enable damping
	m_velLBForDamp :Vec3d := [1.0, 1.0, 0.2];
	
	// max damp
	m_maxDamp :Vec3d := [50, 50, 500];
	
	// distance buffer from joint limit to start damp
	m_limitBufferForDamp :Vec3d :=[20*g_deg2Rad, 20*g_deg2Rad, 0.03];
	
END_VAR

// override this function in each exact controller
METHOD PROTECTED calcCmdJntPos : BOOL
VAR_IN_OUT CONSTANT
	i_endoscopePose : ST_Frame;
	i_masterStatus :ST_MasterStatus;
	i_setupStatus: ST_SetupStatus;
	i_slaveArm :FB_SlaveArm;
END_VAR
m_cmdJntPos[1]:=i_slaveArm.curJntPos[1];
m_cmdJntPos[2]:=i_slaveArm.curJntPos[2];
m_cmdJntPos[3]:=i_slaveArm.curJntPos[3];
IF m_jntOPMode[8] = DriverOPMode_Trq THEN
	m_cmdJntPos[8]:=i_slaveArm.curJntPos[8];
END_IF
IF m_jntOPMode[7] = DriverOPMode_Trq THEN
	m_cmdJntPos[7]:=i_slaveArm.curJntPos[7];
END_IF

m_cmdCartPose:=i_slaveArm.curCartPose;
END_METHOD

// override this function in each exact controller
METHOD PROTECTED calcCmdJntTrq : BOOL
VAR_IN_OUT CONSTANT
	i_endoscopePose : ST_Frame;
	i_masterStatus :ST_MasterStatus;
	i_setupStatus: ST_SetupStatus;
	i_slaveArm :FB_SlaveArm;
END_VAR
VAR
	i :INT;
	dampScale :LREAL;
	limitDis:LREAL;
END_VAR
// set joint torque to zero in default
m_cmdJntTrq := g_zeroVec8d;

// enable endoscope rotation joint if external torque exceed specific value
IF i_slaveArm.instrument.onChipData.m_InstruReadSucceed AND i_slaveArm.instrument.instruType = InstruType_Endoscope AND ABS(i_slaveArm.filtJntCurrent[8]) > 100 THEN
		m_jntOPMode[8]:=DriverOPMode_Trq;
END_IF


// add damp near joint limit
FOR i:=1 TO 3 DO
	IF (i_slaveArm.curJntPos[i] > GVL_SlaveMotorParameters.g_maxDHJntPos[i] - m_limitBufferForDamp[i] AND  i_slaveArm.curJntVel[i]> 0 ) 
		OR (i_slaveArm.curJntPos[i] < GVL_SlaveMotorParameters.g_minDHJntPos[i] + m_limitBufferForDamp[i] AND  i_slaveArm.curJntVel[i]<0 )  THEN
		limitDis := MIN(GVL_SlaveMotorParameters.g_maxDHJntPos[i] - i_slaveArm.curJntPos[i], i_slaveArm.curJntPos[i]-GVL_SlaveMotorParameters.g_minDHJntPos[i]);
		dampScale  :=LIMIT(0, 1-limitDis/m_limitBufferForDamp[i],1);
		m_cmdJntTrq[i]:= -dampScale * m_maxDamp[i] * i_slaveArm.curJntVel[i];
	END_IF
END_FOR

// compute damp
FOR i:=1 TO 3 DO
	IF ABS(i_slaveArm.curJntVel[i]) > m_velLBForDamp[i] THEN 
		dampScale:=LIMIT(0, (ABS(i_slaveArm.curJntVel[i])- m_velLBForDamp[i])/(m_maxAdjustVel[i] - m_velLBForDamp[i]), 1 );
		m_cmdJntTrq[i] :=m_cmdJntTrq[i] -i_slaveArm.curJntVel[i] * m_maxDamp[i] * dampScale;
	END_IF
END_FOR
END_METHOD

METHOD PUBLIC init : BOOL
VAR_IN_OUT CONSTANT
	i_slaveArm	:FB_SlaveArm;
END_VAR
VAR_IN_OUT 
	r_slaveArmCtrlCmd :ST_SlaveArmCtrlCmds;
END_VAR
// check if to hold the command joint position unchanged
m_holdLastCmds := checkToHoldLastCmds(i_slaveArm);

//init
SUPER^.Init(i_slaveArm,r_slaveArmCtrlCmd);


// joint 1/2/3/7 run in torque mode
m_jntOPMode[1]:=DriverOPMode_Trq;
m_jntOPMode[2]:=DriverOPMode_Trq;
m_jntOPMode[3]:=DriverOPMode_Trq;
m_jntOPMode[4]:=DriverOPMode_PosTrq;
m_jntOPMode[5]:=DriverOPMode_PosTrq;
m_jntOPMode[6]:=DriverOPMode_PosTrq;
m_jntOPMode[7]:=DriverOPMode_PosTrq;
m_jntOPMode[8]:=DriverOPMode_PosTrq;

IF i_slaveArm.instrument.onChipData.m_InstruReadSucceed THEN
	IF i_slaveArm.instrument.instruType <> InstruType_Endoscope THEN
		m_jntOPMode[7]:=DriverOPMode_Trq;
	END_IF
END_IF

// update commands to arm
copyCmds(r_slaveArmCtrlCmd);
END_METHOD

END_FUNCTION_BLOCK

// ---- FBs_SlaveControllers/FB_SlaveCtrlMountPanel.TcPOU
// Brief: Mounting Panel
FUNCTION_BLOCK PUBLIC FB_SlaveCtrlMountPanel EXTENDS FB_SlaveArmCtrlBase
VAR_INPUT
END_VAR
VAR_OUTPUT
END_VAR
VAR
	// mount status
	m_mountStatus :INT := 0;
	
	// flag if joint is mounted
	m_jointMounted :ARRAY[1..5] OF BOOL := [5(FALSE)];
	
	// mount motion planning
	m_jntOTG :ARRAY[1..5] OF FB_secOrdTrajFilter;
	m_panelMountVel :LREAL := 2*pi;
	m_panelMountAcc :LREAL := 4*pi;
	
	// joint current threshold which indicate motor is buckled with panel
	m_maxJntCurrent :INT := 180;
	
	// command mount motion
	m_mountStepPos :LREAL := 45.0 * g_deg2Rad;
	m_targetMountPos :Vec5d;
END_VAR

// override this function in each exact controller
METHOD PROTECTED calcCmdJntPos : BOOL
VAR_IN_OUT CONSTANT
	i_endoscopePose : ST_Frame;
	i_masterStatus :ST_MasterStatus;
	i_setupStatus: ST_SetupStatus;
	i_slaveArm :FB_SlaveArm;
END_VAR

VAR 
	i :INT;
	curJntPos :Vec8d;
	jntPosErr :Vec8d;
	cycleNum :LREAL;
END_VAR

curJntPos := i_slaveArm.curJntPos;

CASE m_mountStatus OF
	// To lock joint with panel
	0:
		FOR i:=1 TO 5 DO
			// check joint buckled with panel
			IF ABS(i_slaveArm.filtJntCurrent[i+3])> m_maxJntCurrent THEN 
				m_jointMounted[i]:=TRUE;
				m_targetMountPos[i]:=curJntPos[i+3];
				m_jntOTG[i].init(m_targetMountPos[i], 0,m_panelMountVel, m_panelMountAcc, g_slaveArmCtrlCycleTime);
			END_IF
			
			// set command joint position step
			IF FALSE = m_jointMounted[i] THEN
				m_targetMountPos[i]:=curJntPos[i+3]+m_mountStepPos;
			END_IF
		END_FOR
		
		IF (m_jointMounted[1] AND m_jointMounted[2] AND m_jointMounted[3] AND m_jointMounted[4] AND m_jointMounted[5]) OR m_timePeriod > 5.0 THEN
			m_mountStatus:=1;
		END_IF
	
	// determine zero position
	1:
		FOR i:=1 TO 5 DO
			cycleNum := FLOOR(curJntPos[i+3]/g_2pi);
			m_targetMountPos[i]:=cycleNum* g_2Pi;
		END_FOR
		m_mountStatus :=2;
	
	// move back to zero position
	2:
		m_isFinished:=TRUE;
		FOR i:=1 TO 5 DO
			IF ABS(m_targetMountPos[i]-curJntPos[i+3])>GVL_SlaveControlParameters.g_jntCtrlAngTolHigh THEN
				m_isFinished:=FALSE;
				EXIT;
			END_IF
		END_FOR
END_CASE

// traj plan
FOR i:=1 TO 5 DO
	m_jntOTG[i].run(m_targetMountPos[i],0.0, o_cmdAcc=>m_cmdJntAcc[3+i],o_cmdVel=>m_cmdJntVel[3+i],o_cmdPos=>m_cmdJntPos[i+3]);
END_FOR
END_METHOD

METHOD PUBLIC init : BOOL
VAR_IN_OUT CONSTANT
	i_slaveArm	:FB_SlaveArm;
END_VAR
VAR_IN_OUT 
	r_slaveArmCtrlCmd :ST_SlaveArmCtrlCmds;
END_VAR
VAR
	i : INT;
END_VAR
SUPER^.Init(i_slaveArm,r_slaveArmCtrlCmd);
m_jntOPMode[4] := DriverOPMode_PosTrq;
m_jntOPMode[5] := DriverOPMode_PosTrq;
m_jntOPMode[6] := DriverOPMode_PosTrq;
m_jntOPMode[7] := DriverOPMode_PosTrq;
m_jntOPMode[8] := DriverOPMode_PosTrq;

m_mountStatus:=0;
FOR i:=1 TO 5 DO
	m_targetMountPos[i]:=m_cmdJntPos[i+3];
	m_jntOTG[i].init(m_targetMountPos[i], 0,m_panelMountVel, m_panelMountAcc, g_slaveArmCtrlCycleTime);
	m_jointMounted[i]:=FALSE;
END_FOR

// update commands to arm
copyCmds(r_slaveArmCtrlCmd);
END_METHOD

END_FUNCTION_BLOCK

// ---- FBs_SlaveControllers/FB_SlaveCtrlInstruAutoTest.TcPOU
// Brief: Slave Arm test
FUNCTION_BLOCK PUBLIC FB_SlaveCtrlInstruAutoTest EXTENDS FB_SlaveArmCtrlBase
VAR
											
	m_testStep :INT :=0;
				

	// final target DH joint position and grip angle
	m_targetDHJntPos:Vec3d;
	m_targetGripAng:LREAL;
	m_targetGripForceLevel :LREAL :=0;
	m_targetJntPos :Vec8d;
	
	// interploated command joint position and grip angle 
	m_cmdDHJntPos :Vec6d;
	m_cmdDHJntVel :Vec6d;
	m_cmdGripAng:LREAL;

	// last joint position 
	m_lastCmdJntPos :Vec8d ;
	
	// instrument controller
	m_instruController : FB_BasicInstruControl;
	m_usKnifeController : FB_UltrosonicKnifeControl;
	m_instruCmdJntPos,m_instruCmdJntVel : Vec5d;
	m_instruCmdJntTrq :Vec5d;
	m_maxGripCurrent:LREAL:=350.0;
	m_maxGripCtrlCurrent:LREAL:=540.0;
	m_maxGripCurrentMin:LREAL:=200.0;
	m_maxGripCtrlCurrentMin:LREAL:=400.0;
	
	// OTG
	m_DHJntOTG:ARRAY[1..3] OF FB_secOrdTrajFilter;
	m_gripAngleOTG : FB_secOrdTrajFilter;
	m_jntOTG :ARRAY [1..5] OF FB_secOrdTrajFilter;
	m_maxDHJntVel:Vec3d := [3(2*pi)];
	m_maxDHJntAcc:Vec3d := [3(4*pi)];
	m_maxJntVel:Vec5d := [5(1.57)];
	m_maxJntAcc:Vec5d := [5(3.14)];
	m_testCycles: INT := 0;
	m_instruTestMode: INT := 0;
	iStep: INT;
	m_instruPos: ARRAY [1..60, 1..5] OF LREAL;
	m_openCloseTest: ARRAY [1..60, 1..5] OF LREAL:=
	[0,		0-90,		0,				0,		0,	
	0,		0-90,		0,	     		15,		0,	
	0,		0-90,		0,				30,	    0,	
	0,		0-90,		0,				15,		0,
	0,		0-90,		0,				GVL_InstruTestUIVars.g_maxGripAngle,	    0,
	0,		0-90,		0,				30,	    0,
	0,		0-90,		0,				GVL_InstruTestUIVars.g_minGripAngle,	    100,
	0,		0-90,		0,				0,	    0,
	0,		0-90,		0,				0,	    0,
	0,		0-90,		0,				0,	    0,
	0,		0-90,		0,				0,	    0
	];
	iStep1: INT;
	iStep2: INT;
	m_targetGripAngLast: LREAL;
	m_armIdx:INT;
	m_openGripMoveTest: ARRAY [1..60, 1..5] OF LREAL:=
	[0,		0-90,		0,				0,		                                        0,	
	0,		0-90,		0,	     		GVL_InstruTestUIVars.g_maxGripAngle,		0,	
	0,		0-90,		0,				-90,		 									100,	
	0,		0-90,		60,				-90,											100,	
	0,		0-90,		60,				GVL_InstruTestUIVars.g_maxGripAngle,		0,	
	0,		0-90,		60,				-90,											100,
	0,		0-90,		-60,			-90,											100,
	0,		0-90,		-60,			GVL_InstruTestUIVars.g_maxGripAngle,		0,
	0,		0-90,		-60,			-90,											100,	
	0,		0-90,		0,				-90,											100,	
	0,		90-90,		0,				-90,											100,
	0,		90-90,		0,				GVL_InstruTestUIVars.g_maxGripAngle,		0,
	0,		90-90,		0,				-90,											100,
	0,		-90-90,	0,				-90,											100,
	0,		-90-90,	0,				GVL_InstruTestUIVars.g_maxGripAngle,		0,
	0,		-90-90,	0,				-90,											100,
	0,		0-90,		0,				-90,											100,
	0,		90-90,		60,				-90,											100,
	0,		90-90,		60,	     		GVL_InstruTestUIVars.g_maxGripAngle,		0,	
	0,		90-90,		60,				-90,		 									100,	
	0,		90-90,		-60,			-90,											100,	
	0,		90-90,		-60,			GVL_InstruTestUIVars.g_maxGripAngle,		0,	
	0,		90-90,		-60,			-90,											100,
	0,		-90-90,	-60,			-90,											100,
	0,		-90-90,	-60,			GVL_InstruTestUIVars.g_maxGripAngle,		0,
	0,		-90-90,	-60,			-90,											100,	
	0,		-90-90,	60,				-90,											100,	
	0,		-90-90,	60,				GVL_InstruTestUIVars.g_maxGripAngle,		0,
	0,		-90-90,	60,				-90,											100,
	0,		0-90,		0,				-90,											100,
	0,		0-90,		0,				GVL_InstruTestUIVars.g_maxGripAngle,		0,
	180,	0-90,		60,				GVL_InstruTestUIVars.g_maxGripAngle,		0,
	180,	0-90,		60,				-90,											100,
	180,	0-90,		60,				GVL_InstruTestUIVars.g_maxGripAngle,		0,
	180,	0-90,		-60,			GVL_InstruTestUIVars.g_maxGripAngle,		0,
	180,	0-90,		-60,			-90,											100,
	180,	0-90,		-60,			GVL_InstruTestUIVars.g_maxGripAngle,		0,
	180,	0-90,		0,				GVL_InstruTestUIVars.g_maxGripAngle,		0,
	180,	90-90,		0,				GVL_InstruTestUIVars.g_maxGripAngle,		0,
	180,	90-90,		0,				-90,											100,
	180,	90-90,		0,				GVL_InstruTestUIVars.g_maxGripAngle,		0,
	180,	-90-90,	0,				GVL_InstruTestUIVars.g_maxGripAngle,		0,
	180,	-90-90,	0,				-90,											100,
	180,	-90-90,	0,				GVL_InstruTestUIVars.g_maxGripAngle,		0,
	180,	0-90,		0,				GVL_InstruTestUIVars.g_maxGripAngle,		0,
	180,	90-90,		60,				GVL_InstruTestUIVars.g_maxGripAngle,		0,
	180,	90-90,		60,				-90,											100,
	180,	90-90,		60,				GVL_InstruTestUIVars.g_maxGripAngle,		0,
	180,	90-90,		-60,			GVL_InstruTestUIVars.g_maxGripAngle,		0,
	180,	90-90,		-60,			-90,											100,
	180,	90-90,		-60,			GVL_InstruTestUIVars.g_maxGripAngle,		0,
	180,	-90-90,	-60,			GVL_InstruTestUIVars.g_maxGripAngle,		0,
	180,	-90-90,	-60,			-90,											100,
	180,	-90-90,	-60,			GVL_InstruTestUIVars.g_maxGripAngle,		0,
	180,	-90-90,	60,				GVL_InstruTestUIVars.g_maxGripAngle,		0,
	180,	-90-90,	60,				-90,											100,
	180,	-90-90,	60,				GVL_InstruTestUIVars.g_maxGripAngle,		0,
	0,		0-90,		0,				0,												0,
	0,		0-90,		0,				0,												0,
	0,		0-90,		0,				0,												0
	];
	bstepMove: BOOL;
	fbTonAutoStep: TON;
	fbTime: FB_Timer;
	m_currentNotReached:BOOL;
	fbTonCurrentNotReached:TON;
	bStart: BOOL;
	m_openAngleInitCompensation:LREAL;
	m_GraspingForcepsTest: ARRAY [1..60, 1..5] OF LREAL:=
	[0,		0-90,		0,				0,		                                    0,	
	0,		0-90,		0,	     		GVL_InstruTestUIVars.g_maxGripAngle,		0,	
	0,		0-90,		0,				0,		 									0,	
	0,		0-90,		-60,			0,											0,	
	0,		0-90,		60,				0,											0,	
	0,		0-90,		0,				0,											0,
	0,		-60-90,	0,				0,											0,
	0,		60-90,		0,				0,											0,
	0,		0-90,		0,				0,											0,	
	180,	0-90,		0,				0,											0,	
	180,	0-90,		0,				GVL_InstruTestUIVars.g_maxGripAngle,		0,
	180,	0-90,		0,				0,											0,	
	180,	0-90,		-60,			0,											0,	
	180,	0-90,		60,			    0,											0,	
	180,	0-90,		0,				0,											0,	
	180,	-60-90,	0,				0,											0,	
	180,	60-90,		0,				0,											0,	
	  0,	0-90,		0,				0,											0,	
	-180,	0-90,		0,				0,											0,	 
	-180,	0-90,		0,				GVL_InstruTestUIVars.g_maxGripAngle,		0,	   
	-180,	0-90,		0,				0,											0,	 
	-180,	0-90,		-60,			0,											0,	   
	-180,	0-90,		60,				0,											0,	
	-180,	0-90,		0,				0,											0,	 
    -180,	-60-90,	0,				0,											0,	 
	-180,	60-90,		0,				0,											0,
	0,		0-90,		0,				0,											0,
	0,		0-90,		0,				0,											0,
	0,		0-90,		0,				0,		 										0,
	0,		0-90,		0,				0,		 										0
	];
	m_holdTheNeedleTest: ARRAY [1..60, 1..5] OF LREAL:=
	[0,		0-90,		0,				0,		                                        0,	
	0,		0-90,		0,	     		-60,			0,	
	0,		0-90,		0,				-60,		 									100,	
	0,		0-90,		-60,			-60,											100,	
	0,		0-90,		60,				-60,											100,
	0,		0-90,		0,				-60,		 									100,	
	0,		-60-90,	0,				-60,		 									100,	
	0,		60-90,		0,				-60,		 									100,
	0,		0-90,		0,				-60,		 									100,
	180,	0-90,		0,				-60,		 									100,
	180,	0-90,		-60,			-60,		 									100,
	180,	0-90,		60,				-60,		 									100,
	180,	0-90,		0,				-60,		 									100,
	180,	-60-90,	0,				-60,		 									100,
	180,	60-90,		0,				-60,		 									100,
	180,	0-90,		0,				-60,		 									100,
	-180,	0-90,		0,				-60,		 									100,
	-180,	0-90,		-60,			-60,		 									100,
	-180,	0-90,		60,				-60,		 									100,
	-180,	0-90,		0,				-60,		 									100,
	-180,	-60-90,	0,				-60,		 									100,
	-180,	60-90,		0,				-60,		 									100,
	-180,	0-90,		0,				-60,		 									100,
	0,		0-90,		0,				0,		 										0,
	0,		0-90,		0,				0,		 										0,
	0,		0-90,		0,				0,		 										0,
	0,		0-90,		0,				0,		 										0
	];
	
	// instrument tyep
	m_instruType : E_InstrumentType;
	m_openGripMoveTestCautery: ARRAY [1..60, 1..5] OF LREAL:=
	[0,		0-90,		0,				0,		                                        0,	
	0,		0-90,		0,	     		GVL_InstruTestUIVars.g_maxGripAngle,		0,	
	0,		0-90,		0,				-90,		 									100,	
	0,		0-90,		60,				-90,											100,	
	0,		0-90,		60,				GVL_InstruTestUIVars.g_maxGripAngle,		0,	
	0,		0-90,		60,				-90,											100,
	0,		0-90,		-60,			-90,											100,
	0,		0-90,		-60,			GVL_InstruTestUIVars.g_maxGripAngle,		0,
	0,		0-90,		-60,			-90,											100,	
	0,		0-90,		0,				-90,											100,	
	0,		90-90-20,		0,				-90,											100,
	0,		90-90-20,		0,				GVL_InstruTestUIVars.g_maxGripAngle,		0,
	0,		90-90-20,		0,				-90,											100,
	0,		-90-90+20,	0,				-90,											100,
	0,		-90-90+20,	0,				GVL_InstruTestUIVars.g_maxGripAngle,		0,
	0,		-90-90+20,	0,				-90,											100,
	0,		0-90,		0,				-90,											100,
	0,		90-90-20,		60,				-90,											100,
	0,		90-90-20,		60,	     		GVL_InstruTestUIVars.g_maxGripAngle,		0,	
	0,		90-90-20,		60,				-90,		 									100,	
	0,		90-90-20,		-60,			-90,											100,	
	0,		90-90-20,		-60,			GVL_InstruTestUIVars.g_maxGripAngle,		0,	
	0,		90-90-20,		-60,			-90,											100,
	0,		-90-90+20,	-60,			-90,											100,
	0,		-90-90+20,	-60,			GVL_InstruTestUIVars.g_maxGripAngle,		0,
	0,		-90-90+20,	-60,			-90,											100,	
	0,		-90-90+20,	60,				-90,											100,	
	0,		-90-90+20,	60,				GVL_InstruTestUIVars.g_maxGripAngle,		0,
	0,		-90-90+20,	60,				-90,											100,
	0,		0-90,		0,				-90,											100,
	0,		0-90,		0,				GVL_InstruTestUIVars.g_maxGripAngle,		0,
	180,	0-90,		60,				GVL_InstruTestUIVars.g_maxGripAngle,		0,
	180,	0-90,		60,				-90,											100,
	180,	0-90,		60,				GVL_InstruTestUIVars.g_maxGripAngle,		0,
	180,	0-90,		-60,			GVL_InstruTestUIVars.g_maxGripAngle,		0,
	180,	0-90,		-60,			-90,											100,
	180,	0-90,		-60,			GVL_InstruTestUIVars.g_maxGripAngle,		0,
	180,	0-90,		0,				GVL_InstruTestUIVars.g_maxGripAngle,		0,
	180,	90-90-20,		0,				GVL_InstruTestUIVars.g_maxGripAngle,		0,
	180,	90-90-20,		0,				-90,											100,
	180,	90-90-20,		0,				GVL_InstruTestUIVars.g_maxGripAngle,		0,
	180,	-90-90+20,	0,				GVL_InstruTestUIVars.g_maxGripAngle,		0,
	180,	-90-90+20,	0,				-90,											100,
	180,	-90-90+20,	0,				GVL_InstruTestUIVars.g_maxGripAngle,		0,
	180,	0-90,		0,				GVL_InstruTestUIVars.g_maxGripAngle,		0,
	180,	90-90-20,		60,				GVL_InstruTestUIVars.g_maxGripAngle,		0,
	180,	90-90-20,		60,				-90,											100,
	180,	90-90-20,		60,				GVL_InstruTestUIVars.g_maxGripAngle,		0,
	180,	90-90-20,		-60,			GVL_InstruTestUIVars.g_maxGripAngle,		0,
	180,	90-90-20,		-60,			-90,											100,
	180,	90-90-20,		-60,			GVL_InstruTestUIVars.g_maxGripAngle,		0,
	180,	-90-90+20,	-60,			GVL_InstruTestUIVars.g_maxGripAngle,		0,
	180,	-90-90+20,	-60,			-90,											100,
	180,	-90-90+20,	-60,			GVL_InstruTestUIVars.g_maxGripAngle,		0,
	180,	-90-90+20,	60,				GVL_InstruTestUIVars.g_maxGripAngle,		0,
	180,	-90-90+20,	60,				-90,											100,
	180,	-90-90+20,	60,				GVL_InstruTestUIVars.g_maxGripAngle,		0,
	0,		0-90,		0,				0,												0,
	0,		0-90,		0,				0,												0,
	0,		0-90,		0,				0,												0
	];
	m_setTestCycles: INT;
	m_openGripMoveTestMode: ARRAY [1..60, 1..5] OF LREAL:=
	[0,		0-90,		0,				0,		                                        0,	
	0,		0-90,		0,	     		GVL_InstruTestUIVars.g_maxGripAngle,		0,	
	0,		0-90,		0,				-90,		 									100,	
	0,		0-90,		60,				-90,											100,	
	0,		0-90,		60,				GVL_InstruTestUIVars.g_maxGripAngle,		0,	
	0,		0-90,		60,				-90,											100,
	0,		0-90,		-60,			-90,											100,
	0,		0-90,		-60,			GVL_InstruTestUIVars.g_maxGripAngle,		0,
	0,		0-90,		-60,			-90,											100,	
	0,		0-90,		0,				-90,											100,	
	0,		90-90,		0,				-90,											100,
	0,		90-90,		0,				GVL_InstruTestUIVars.g_maxGripAngle,		0,
	0,		90-90,		0,				-90,											100,
	0,		-90-90,	0,				-90,											100,
	0,		-90-90,	0,				GVL_InstruTestUIVars.g_maxGripAngle,		0,
	0,		-90-90,	0,				-90,											100,
	0,		0-90,		0,				-90,											100,
	0,		90-90,		60,				-90,											100,
	0,		90-90,		60,	     		GVL_InstruTestUIVars.g_maxGripAngle,		0,	
	0,		90-90,		60,				-90,		 									100,	
	0,		90-90,		-60,			-90,											100,	
	0,		90-90,		-60,			GVL_InstruTestUIVars.g_maxGripAngle,		0,	
	0,		90-90,		-60,			-90,											100,
	0,		-90-90,	-60,			-90,											100,
	0,		-90-90,	-60,			GVL_InstruTestUIVars.g_maxGripAngle,		0,
	0,		-90-90,	-60,			-90,											100,	
	0,		-90-90,	60,				-90,											100,	
	0,		-90-90,	60,				GVL_InstruTestUIVars.g_maxGripAngle,		0,
	0,		-90-90,	60,				-90,											100,
	0,		0-90,		0,				-90,											100,
	0,		0-90,		0,				GVL_InstruTestUIVars.g_maxGripAngle,		0,
	180,	0-90,		60,				GVL_InstruTestUIVars.g_maxGripAngle,		0,
	180,	0-90,		60,				-90,											100,
	180,	0-90,		60,				GVL_InstruTestUIVars.g_maxGripAngle,		0,
	180,	0-90,		-60,			GVL_InstruTestUIVars.g_maxGripAngle,		0,
	180,	0-90,		-60,			-90,											100,
	180,	0-90,		-60,			GVL_InstruTestUIVars.g_maxGripAngle,		0,
	180,	0-90,		0,				GVL_InstruTestUIVars.g_maxGripAngle,		0,
	180,	90-90,		0,				GVL_InstruTestUIVars.g_maxGripAngle,		0,
	180,	90-90,		0,				-90,											100,
	180,	90-90,		0,				GVL_InstruTestUIVars.g_maxGripAngle,		0,
	180,	-90-90,	0,				GVL_InstruTestUIVars.g_maxGripAngle,		0,
	180,	-90-90,	0,				-90,											100,
	180,	-90-90,	0,				GVL_InstruTestUIVars.g_maxGripAngle,		0,
	180,	0-90,		0,				GVL_InstruTestUIVars.g_maxGripAngle,		0,
	180,	90-90,		60,				GVL_InstruTestUIVars.g_maxGripAngle,		0,
	180,	90-90,		60,				-90,											100,
	180,	90-90,		60,				GVL_InstruTestUIVars.g_maxGripAngle,		0,
	180,	90-90,		-60,			GVL_InstruTestUIVars.g_maxGripAngle,		0,
	180,	90-90,		-60,			-90,											100,
	180,	90-90,		-60,			GVL_InstruTestUIVars.g_maxGripAngle,		0,
	180,	-90-90,	-60,			GVL_InstruTestUIVars.g_maxGripAngle,		0,
	180,	-90-90,	-60,			-90,											100,
	180,	-90-90,	-60,			GVL_InstruTestUIVars.g_maxGripAngle,		0,
	180,	-90-90,	60,				GVL_InstruTestUIVars.g_maxGripAngle,		0,
	180,	-90-90,	60,				-90,											100,
	180,	-90-90,	60,				GVL_InstruTestUIVars.g_maxGripAngle,		0,
	0,		0-90,		0,				0,												0,
	0,		0-90,		0,				0,												0,
	0,		0-90,		0,				0,												0
	];
END_VAR

METHOD PROTECTED calcCmdJntPos : BOOL
VAR_IN_OUT CONSTANT
	i_endoscopePose : ST_Frame;
	i_masterStatus :ST_MasterStatus;
	i_setupStatus: ST_SetupStatus;
	i_slaveArm :FB_SlaveArm;
END_VAR

VAR 
	i:INT :=0;

END_VAR
GVL_InstruTestUIVars.g_curTestCycles:=m_testCycles;
IF GVL_InstruTestUIVars.g_autoTestStart THEN 
	bStart:=TRUE;
	GVL_InstruTestUIVars.g_autoTestStart:=FALSE;
END_IF
IF GVL_InstruTestUIVars.g_autoTestStop THEN 
	m_isFinished := TRUE;
	GVL_InstruTestUIVars.g_autoTestStop:=FALSE;
END_IF
IF bStart AND NOT GVL_InstruTestUIVars.g_autoTestPause THEN 
	instruTestMode(i_slaveArm);
END_IF
(*
IF ABS( m_targetGripAngLast-m_targetGripAng)>0.0001  THEN
  IF  m_targetGripAngLast-m_targetGripAng<0.0001   THEN
	  m_targetGripAng:=m_targetGripAng+m_openAngleInitCompensation*g_deg2rad;
  ELSE
	  m_targetGripAng:=m_targetGripAng;
  END_IF                       
END_IF
m_targetGripAngLast:=m_targetGripAng;
*)
//CurrentDetection
IF GVL_InstruTestUIVars.g_funcCurrentDetection THEN	
	IF ABS (i_slaveArm.filtJntCurrent[1] -GVL_InstruTestUIVars.g_actualRatedCurrent[4])>5 AND 
	   ABS (i_slaveArm.filtJntCurrent[2] -GVL_InstruTestUIVars.g_actualRatedCurrent[5])>5 THEN
		m_currentNotReached:=FALSE;
	ELSE 
		m_currentNotReached:=TRUE;
	END_IF	
	fbTonCurrentNotReached(IN:= m_currentNotReached, PT:= T#60S, Q=> , ET=> );
	
	IF fbTonCurrentNotReached.Q THEN
		m_isFinished := TRUE;
		m_currentNotReached:=FALSE;
	END_IF
END_IF
//TIME
fbTime.timer(bStart:=TRUE,uiTimeHour=>GVL_InstruTestUIVars.g_testTimeHour,
					uiTimeMinute=>GVL_InstruTestUIVars.g_testTimeMinute,
					uiTimeSecond=>GVL_InstruTestUIVars.g_testTimeSecond);
// run OTG
FOR i:=1 TO 3  DO
	m_DHJntOTG[i].run(m_targetDHJntPos[i],0.0, o_cmdAcc=>,o_cmdVel=>m_cmdDHJntVel[i],o_cmdPos=> m_cmdDHJntPos[i+3]);
END_FOR
m_gripAngleOTG.run(m_targetGripAng,0.0, o_cmdAcc=>,o_cmdVel=>,o_cmdPos=>m_cmdGripAng);
//FOR i:=1 TO 3  DO
//	m_cmdDHJntPos[i+3] := m_targetDHJntPos[i];
//	m_cmdGripAng := m_targetGripAng;
//END_FOR

// calculate target motor joint position from DH joint position
i_slaveArm.instrument.instruIK(m_cmdDHJntPos,m_cmdGripAng, o_jntPos=>m_cmdJntPos);
//FOR i:=1 TO 5 DO
//	m_jntOTG[i].run(m_targetJntPos[i+3],0.0, o_cmdAcc=>,o_cmdVel=>m_cmdJntVel[i+3],o_cmdPos=> m_cmdJntPos[i+3]);
//END_FOR


// command velocity
vecSub(m_cmdJntPos, m_lastCmdJntPos, m_cmdJntVel);
vecSelfMultiNum(m_cmdJntVel, g_slaveArmCtrlFreq);
m_lastCmdJntPos:=m_cmdJntPos;
END_METHOD

// override this function in each exact controller
METHOD PROTECTED calcCmdJntTrq : BOOL
VAR_IN_OUT CONSTANT
	i_endoscopePose : ST_Frame;
	i_masterStatus :ST_MasterStatus;
	i_setupStatus: ST_SetupStatus;
	i_slaveArm :FB_SlaveArm;
END_VAR

VAR 
	nullspaceMat :Mat7d;
	ctrlTrq : Vec7d;
	i : int ;
END_VAR
// set joint torque to zero in default
m_cmdJntTrq := g_zeroVec8d;

// instrument joint control
FOR i:=1 TO 5 DO 
	m_instruCmdJntPos[i]:=m_cmdJntPos[i+3];
	m_instruCmdJntVel[i]:=m_cmdJntVel[i+3];
END_FOR

IF i_slaveArm.instrument.instruType = InstruType_UltrasoundKnifeS OR i_slaveArm.instrument.instruType = InstruType_UltrasoundKnifeU THEN
	m_usKnifeController.run(m_instruCmdJntPos,m_instruCmdJntVel, m_targetGripForceLevel, i_slaveArm, o_cmdJntTrq=>m_instruCmdJntTrq);
ELSE
	m_instruController.run(m_instruCmdJntPos,m_instruCmdJntVel, m_cmdDHJntPos[6], m_cmdDHJntVel[6], m_targetGripForceLevel, i_slaveArm, o_cmdJntTrq=>m_instruCmdJntTrq);
END_IF

FOR i:=1 TO 5 DO
	m_cmdJntTrq[i+3]:=m_instruCmdJntTrq[i];
END_FOR
END_METHOD

PROPERTY getTestMode : INT
GET
getTestMode:=m_instruTestMode;
END_GET
END_PROPERTY

METHOD PUBLIC init : BOOL
VAR_IN_OUT CONSTANT
	i_slaveArm	:FB_SlaveArm;
END_VAR
VAR_IN_OUT 
	r_slaveArmCtrlCmd :ST_SlaveArmCtrlCmds;
END_VAR

VAR
	i:int;
END_VAR
SUPER^.Init(i_slaveArm,r_slaveArmCtrlCmd);
m_lastCmdJntPos:=m_cmdJntPos;
IF GVL_InstruTestUIVars.g_testMode=3 THEN
	m_jntOPMode[1] := DriverOPMode_PosTrq;
	m_jntOPMode[2] := DriverOPMode_PosTrq;
	m_jntOPMode[3] := DriverOPMode_PosTrq;
	m_jntOPMode[4] := DriverOPMode_Pos;
	m_jntOPMode[5] := DriverOPMode_Pos;
	m_jntOPMode[6] := DriverOPMode_Pos;
	m_jntOPMode[7] := DriverOPMode_Pos;
	m_jntOPMode[8] := DriverOPMode_Pos;
ELSE
	m_jntOPMode[1] := DriverOPMode_PosTrq;
	m_jntOPMode[2] := DriverOPMode_PosTrq;
	m_jntOPMode[3] := DriverOPMode_PosTrq;
	m_jntOPMode[4] := DriverOPMode_Trq;
	m_jntOPMode[5] := DriverOPMode_Trq;
	m_jntOPMode[6] := DriverOPMode_Trq;
	m_jntOPMode[7] := DriverOPMode_Trq;
	m_jntOPMode[8] := DriverOPMode_Trq;
END_IF
m_armIdx:=i_slaveArm.armIdx;
fbTime.init();
GVL_InstruTestUIVars.g_autoTestStart:=FALSE;
GVL_InstruTestUIVars.g_autoTestStop:=FALSE;
bStart:=FALSE;
IF GVL_InstruTestUIVars.g_testCycles=0 THEN
	GVL_InstruTestUIVars.g_testCycles:=1;
END_IF
m_instruTestMode := GVL_InstruTestUIVars.g_testMode;  //m_isSingleFinger
IF m_instruTestMode=2 OR m_instruTestMode=3  THEN
	IF i_slaveArm.instrument.onChipData.m_InstruReadSucceed AND i_slaveArm.m_instrument.instruTypeInfo.m_isSingleFinger  THEN
		m_instruTestMode := GVL_InstruTestUIVars.g_testMode+10;
	END_IF
END_IF
m_testStep := 0;
m_testCycles := 1;
m_cmdDHJntPos :=i_slaveArm.curDHJntPos;
m_cmdDHJntVel :=g_zeroVec6d;
m_targetGripAng := i_slaveArm.curGripAngle;
m_targetDHJntPos[1] := i_slaveArm.curDHJntPos[4];
m_targetDHJntPos[2] := i_slaveArm.curDHJntPos[5];
m_targetDHJntPos[3] := i_slaveArm.curDHJntPos[6];


// init instrument controller
IF m_instruTestMode=3  THEN
	m_instruController.init(i_slaveArm,m_maxGripCurrentMin,m_maxGripCtrlCurrentMin);
ELSE
	m_instruController.init(i_slaveArm,m_maxGripCurrent,m_maxGripCtrlCurrent);
END_IF
m_usKnifeController.init(i_slaveArm);
m_instruType := i_slaveArm.instrument.instruType;


FOR i:=1 TO 3  DO
	m_DHJntOTG[i].init(m_cmdDHJntPos[i+3], 0, m_maxDHJntVel[i], m_maxDHJntAcc[i], g_slaveArmCtrlCycleTime);
END_FOR

m_gripAngleOTG.init(m_targetGripAng, 0, m_maxDHJntVel[1], m_maxDHJntAcc[1], g_slaveArmCtrlCycleTime);

FOR i := 1 TO 5 DO
	m_targetJntPos[i] := i_slaveArm.curJntPos[i];
	m_jntOTG[i].init(m_cmdJntPos[i+3], 0, m_maxJntVel[i], m_maxJntAcc[i], g_slaveArmCtrlCycleTime);
END_FOR
// update commands to arm
copyCmds(r_slaveArmCtrlCmd);


iStep:=5;
END_METHOD

PROPERTY InstruBacklash : Vec5d
GET
IF m_instruType = InstruType_UltrasoundKnifeS OR m_instruType = InstruType_UltrasoundKnifeU THEN
	instruBacklash := g_zeroVec5d;
ELSE
	instruBacklash := m_instruController.m_jntBacklash;
END_IF
END_GET
END_PROPERTY

METHOD instruTestMode : BOOL
VAR_IN_OUT CONSTANT
	i_slaveArm :FB_SlaveArm;
END_VAR
VAR
	i:INT;
END_VAR
CASE m_instruTestMode OF
	1:
		m_testStep := LIMIT(0,m_testStep, 9);
		m_instruPos:=m_openCloseTest;
		iStep1:=7;
		iStep2:=6;
		m_setTestCycles:=GVL_InstruTestUIVars.g_testCycles;
	2:
		m_testStep := LIMIT(0,m_testStep, 60);
		m_instruPos:=m_openGripMoveTest;
		iStep1:=58;
		iStep2:=57;
		m_setTestCycles:=GVL_InstruTestUIVars.g_testCycles;
	3:
		m_testStep := LIMIT(0,m_testStep, 60);
		m_instruPos:=m_openGripMoveTestMode;
		iStep1:=58;
		iStep2:=57;
		m_setTestCycles:=GVL_InstruTestUIVars.g_testCycles;
	4:
		m_testStep := LIMIT(0,m_testStep, 29);
		m_instruPos:=m_GraspingForcepsTest;
		iStep1:=27;
		iStep2:=26;
		m_setTestCycles:=GVL_InstruTestUIVars.g_testCycles;
	5:
		m_testStep := LIMIT(0,m_testStep, 26);
		m_instruPos:=m_holdTheNeedleTest;
		iStep1:=24;
		iStep2:=23;
		m_setTestCycles:=GVL_InstruTestUIVars.g_testCycles;
	12:
		m_testStep := LIMIT(0,m_testStep, 60);
		m_instruPos:=m_openGripMoveTestCautery;
		iStep1:=58;
		iStep2:=57;
		m_setTestCycles:=GVL_InstruTestUIVars.g_testCycles;

	13:
		m_testStep := LIMIT(0,m_testStep, 60);
		m_instruPos:=m_openGripMoveTestCautery;
		iStep1:=58;
		iStep2:=57;
		m_setTestCycles:=GVL_InstruTestUIVars.g_testCycles;
	ELSE
		RETURN;
END_CASE
bstepMove:=TRUE;
fbTonAutoStep(IN:=iStep=15 , PT:= T#0.1S, Q=> , ET=> );
GVL_InstruTestUIVars.g_testStep:=m_testStep+1;
CASE iStep OF
	0:;
	5:  
		FOR i:=1 TO 3 BY 1 DO
			m_targetDHJntPos[i] := m_instruPos[m_testStep+1, i]*g_deg2rad;
		END_FOR
		m_targetGripAng := m_instruPos[m_testStep+1, 4]*g_deg2rad;
		m_targetGripForceLevel:=m_instruPos[m_testStep+1, 5];
		IF m_instruTestMode=12 OR m_instruTestMode=13 THEN
			m_targetGripAng :=0;
			m_targetGripForceLevel:=0;
		END_IF
		IF m_targetGripForceLevel>0 AND m_instruTestMode = 1  THEN
			
			m_targetGripAng:=GVL_InstruTestUIVars.g_minGripAngle*g_deg2rad;
		END_IF
		m_targetGripForceLevel:=0;
		
		bstepMove:=FALSE;
		iStep:=10;
	10: 
		IF ABS(m_cmdDHJntPos[4]-m_targetDHJntPos[1])< g_jntCtrlAngTolLow 
		AND ABS(m_cmdDHJntPos[5]-m_targetDHJntPos[2])< g_jntCtrlAngTolLow 	
		AND ABS(m_cmdDHJntPos[6]-m_targetDHJntPos[3])< g_jntCtrlAngTolLow 
		AND ABS(m_cmdGripAng- m_targetGripAng)< g_jntCtrlAngTolLow 
		AND bstepMove  THEN
		    iStep:=15;
	    END_IF
	15: 
	    IF fbTonAutoStep.Q THEN
	    	iStep:=20;
	    END_IF
	20: 
		m_testStep:=m_testStep+1;
		iStep:=5;
		IF m_testStep =iStep1 THEN
			m_testCycles:=m_testCycles+1;
			m_testStep := 0;
		END_IF

		IF m_testCycles>=m_setTestCycles+1 THEN
			m_testCycles:=m_testCycles-1;
			iStep:=25;
		END_IF

	25: 
	    m_testStep:=iStep2+1;
		FOR i:=1 TO 3 BY 1 DO
			m_targetDHJntPos[i] := m_instruPos[m_testStep+1, i]*g_deg2rad;
		END_FOR
        m_targetGripAng := m_instruPos[m_testStep+1, 4]*g_deg2rad;
        m_targetGripForceLevel:=m_instruPos[m_testStep+1, 5];
//		m_testStep:=iStep2+2;
		iStep:=30;
    30: IF ABS(m_cmdDHJntPos[4]-m_targetDHJntPos[1])< g_jntCtrlAngTolLow 
		AND ABS(m_cmdDHJntPos[5]-m_targetDHJntPos[2])< g_jntCtrlAngTolLow 
		AND ABS(m_cmdDHJntPos[6]-m_targetDHJntPos[3])< g_jntCtrlAngTolLow 
		AND ABS(m_cmdGripAng- m_targetGripAng)< g_jntCtrlAngTolLow THEN
		    iStep:=35;
	    END_IF
	35: 
	    m_isFinished := TRUE;
		iStep:=0;
END_CASE
END_METHOD

END_FUNCTION_BLOCK

// ---- FBs_SlaveControllers/FB_SlaveCtrlInstruVerify.TcPOU
// Brief: Slave Arm test
FUNCTION_BLOCK PUBLIC FB_SlaveCtrlInstruVerify EXTENDS FB_SlaveArmCtrlBase
VAR
											
	m_testStep :INT :=0;
				

	// final target DH joint position and grip angle
	m_targetDHJntPos:Vec3d;
	m_targetGripAng:LREAL;
	m_targetGripForceLevel :LREAL :=0;
	
	// interploated command joint position and grip angle 
	m_cmdDHJntPos :Vec6d;
	m_cmdDHJntVel :Vec6d;
	m_cmdGripAng:LREAL;

	// last joint position 
	m_lastCmdJntPos :Vec8d ;
	
	// instrument controller
	m_instruController : FB_BasicInstruControl;
	m_usKnifeController : FB_UltrosonicKnifeControl;
	m_instruCmdJntPos,m_instruCmdJntVel : Vec5d;
	m_instruCmdJntTrq :Vec5d;

	// instrument type
	m_instruType : E_InstrumentType;
	m_maxGripCurrent:LREAL:=350.0;
	m_maxGripCtrlCurrent:LREAL:=540.0;
	
	// OTG
	m_DHJntOTG:ARRAY[1..3] OF FB_secOrdTrajFilter;
	m_gripAngleOTG : FB_secOrdTrajFilter;
	m_maxJntVel:Vec3d := [3(8.0)];
	m_maxJntAcc:Vec3d := [3(50.0)];
	m_testCycles: INT := 0;
	m_instruTestMode: INT := 0;
	iStep: INT;
	m_instruPos: ARRAY [1..60, 1..5] OF LREAL;
	iStep1: INT;
	iStep2: INT;
	m_targetGripAngLast: LREAL;
	m_armIdx:INT;
	bstepMove: BOOL;
	fbTime: FB_Timer;
	m_openAngleInitCompensation:LREAL;
	m_openCloseTest: ARRAY [1..60, 1..5] OF LREAL:=
	[0,		0-90,		0,				0,		0,	
	0,		0-90,		0,	     		15,		0,	
	0,		0-90,		0,				30,	    0,	
	0,		0-90,		0,				15,		0,
	0,		0-90,		0,				GVL_InstruTestUIVars.g_maxGripAngle,	    0,
	0,		0-90,		0,				30,	    0,
	0,		0-90,		0,				GVL_InstruTestUIVars.g_minGripAngle,	    100,
	0,		0-90,		0,				0,	    0
	];
	m_openGripMoveTest: ARRAY [1..60, 1..5] OF LREAL:=
	[0,		0-90,		0,				0,		                                        0,	
	0,		0-90,		0,	     		GVL_InstruTestUIVars.g_maxGripAngle,		0,	
	0,		0-90,		0,				-90,		 									0,	
	0,		0-90,		60,				-90,											0,	
	0,		0-90,		60,				GVL_InstruTestUIVars.g_maxGripAngle,		0,	
	0,		0-90,		60,				-90,											0,
	0,		0-90,		-60,			-90,											0,
	0,		0-90,		-60,			GVL_InstruTestUIVars.g_maxGripAngle,		0,
	0,		0-90,		-60,			-90,											0,	
	0,		0-90,		0,				-90,											0,	
	0,		90-90,		0,				-90,											0,
	0,		90-90,		0,				GVL_InstruTestUIVars.g_maxGripAngle,		0,
	0,		90-90,		0,				-90,											0,
	0,		-90-90,	0,				-90,											0,
	0,		-90-90,	0,				GVL_InstruTestUIVars.g_maxGripAngle,		0,
	0,		-90-90,	0,				-90,											0,
	0,		0-90,		0,				-90,											0,
	0,		90-90,		60,				-90,											0,
	0,		90-90,		60,	     		GVL_InstruTestUIVars.g_maxGripAngle,		0,	
	0,		90-90,		60,				-90,		 									0,	
	0,		90-90,		-60,			-90,											0,	
	0,		90-90,		-60,			GVL_InstruTestUIVars.g_maxGripAngle,		0,	
	0,		90-90,		-60,			-90,											0,
	0,		-90-90,	-60,			-90,											0,
	0,		-90-90,	-60,			GVL_InstruTestUIVars.g_maxGripAngle,		0,
	0,		-90-90,	-60,			-90,											0,	
	0,		-90-90,	60,				-90,											0,	
	0,		-90-90,	60,				GVL_InstruTestUIVars.g_maxGripAngle,		0,
	0,		-90-90,	60,				-90,											0,
	0,		0-90,		0,				-90,											0,
	0,		0-90,		0,				GVL_InstruTestUIVars.g_maxGripAngle,		0,
	180,	0-90,		60,				GVL_InstruTestUIVars.g_maxGripAngle,		0,
	180,	0-90,		60,				-90,											0,
	180,	0-90,		60,				GVL_InstruTestUIVars.g_maxGripAngle,		0,
	180,	0-90,		-60,			GVL_InstruTestUIVars.g_maxGripAngle,		0,
	180,	0-90,		-60,			-90,											0,
	180,	0-90,		-60,			GVL_InstruTestUIVars.g_maxGripAngle,		0,
	180,	0-90,		0,				GVL_InstruTestUIVars.g_maxGripAngle,		0,
	180,	90-90,		0,				GVL_InstruTestUIVars.g_maxGripAngle,		0,
	180,	90-90,		0,				-90,											0,
	180,	90-90,		0,				GVL_InstruTestUIVars.g_maxGripAngle,		0,
	180,	-90-90,	0,				GVL_InstruTestUIVars.g_maxGripAngle,		0,
	180,	-90-90,	0,				-90,											0,
	180,	-90-90,	0,				GVL_InstruTestUIVars.g_maxGripAngle,		0,
	180,	0-90,		0,				GVL_InstruTestUIVars.g_maxGripAngle,		0,
	180,	90-90,		60,				GVL_InstruTestUIVars.g_maxGripAngle,		0,
	180,	90-90,		60,				-90,											0,
	180,	90-90,		60,				GVL_InstruTestUIVars.g_maxGripAngle,		0,
	180,	90-90,		-60,			GVL_InstruTestUIVars.g_maxGripAngle,		0,
	180,	90-90,		-60,			-90,											0,
	180,	90-90,		-60,			GVL_InstruTestUIVars.g_maxGripAngle,		0,
	180,	-90-90,	-60,			GVL_InstruTestUIVars.g_maxGripAngle,		0,
	180,	-90-90,	-60,			-90,											0,
	180,	-90-90,	-60,			GVL_InstruTestUIVars.g_maxGripAngle,		0,
	180,	-90-90,	60,				GVL_InstruTestUIVars.g_maxGripAngle,		0,
	180,	-90-90,	60,				-90,											0,
	180,	-90-90,	60,				GVL_InstruTestUIVars.g_maxGripAngle,		0,
	0,		0-90,		0,				0,												0
	];
	m_tiredTest: ARRAY [1..60, 1..5] OF LREAL:=
	[0,		0-90,		0,				0,		                                        0,	
	0,		0-90,		0,	     		GVL_InstruTestUIVars.g_maxGripAngle,		0,	
	0,		0-90,		0,				-90,		 									0,	
	0,		0-90,		60,				-90,											0,	
	0,		0-90,		60,				GVL_InstruTestUIVars.g_maxGripAngle,		0,	
	0,		0-90,		60,				-90,											0,
	0,		0-90,		-60,			-90,											0,
	0,		0-90,		-60,			GVL_InstruTestUIVars.g_maxGripAngle,		0,
	0,		0-90,		-60,			-90,											0,	
	0,		0-90,		0,				-90,											0,	
	0,		90-90,		0,				-90,											0,
	0,		90-90,		0,				GVL_InstruTestUIVars.g_maxGripAngle,		0,
	0,		90-90,		0,				-90,											0,
	0,		-90-90,	0,				-90,											0,
	0,		-90-90,	0,				GVL_InstruTestUIVars.g_maxGripAngle,		0,
	0,		-90-90,	0,				-90,											0,
	0,		0-90,		0,				-90,											0,
	0,		90-90,		60,				-90,											0,
	0,		90-90,		60,	     		GVL_InstruTestUIVars.g_maxGripAngle,		0,	
	0,		90-90,		60,				-90,		 									0,	
	0,		90-90,		-60,			-90,											0,	
	0,		90-90,		-60,			GVL_InstruTestUIVars.g_maxGripAngle,		0,	
	0,		90-90,		-60,			-90,											0,
	0,		-90-90,	-60,			-90,											0,
	0,		-90-90,	-60,			GVL_InstruTestUIVars.g_maxGripAngle,		0,
	0,		-90-90,	-60,			-90,											0,	
	0,		-90-90,	60,				-90,											0,	
	0,		-90-90,	60,				GVL_InstruTestUIVars.g_maxGripAngle,		0,
	0,		-90-90,	60,				-90,											0,
	0,		0-90,		0,				-90,											0,
	0,		0-90,		0,				GVL_InstruTestUIVars.g_maxGripAngle,		0,
	180,	0-90,		60,				GVL_InstruTestUIVars.g_maxGripAngle,		0,
	180,	0-90,		60,				-90,											0,
	180,	0-90,		60,				GVL_InstruTestUIVars.g_maxGripAngle,		0,
	180,	0-90,		-60,			GVL_InstruTestUIVars.g_maxGripAngle,		0,
	180,	0-90,		-60,			-90,											0,
	180,	0-90,		-60,			GVL_InstruTestUIVars.g_maxGripAngle,		0,
	180,	0-90,		0,				GVL_InstruTestUIVars.g_maxGripAngle,		0,
	180,	90-90,		0,				GVL_InstruTestUIVars.g_maxGripAngle,		0,
	180,	90-90,		0,				-90,											0,
	180,	90-90,		0,				GVL_InstruTestUIVars.g_maxGripAngle,		0,
	180,	-90-90,	0,				GVL_InstruTestUIVars.g_maxGripAngle,		0,
	180,	-90-90,	0,				-90,											0,
	180,	-90-90,	0,				GVL_InstruTestUIVars.g_maxGripAngle,		0,
	180,	0-90,		0,				GVL_InstruTestUIVars.g_maxGripAngle,		0,
	180,	90-90,		60,				GVL_InstruTestUIVars.g_maxGripAngle,		0,
	180,	90-90,		60,				-90,											0,
	180,	90-90,		60,				GVL_InstruTestUIVars.g_maxGripAngle,		0,
	180,	90-90,		-60,			GVL_InstruTestUIVars.g_maxGripAngle,		0,
	180,	90-90,		-60,			-90,											0,
	180,	90-90,		-60,			GVL_InstruTestUIVars.g_maxGripAngle,		0,
	180,	-90-90,	-60,			GVL_InstruTestUIVars.g_maxGripAngle,		0,
	180,	-90-90,	-60,			-90,											0,
	180,	-90-90,	-60,			GVL_InstruTestUIVars.g_maxGripAngle,		0,
	180,	-90-90,	60,				GVL_InstruTestUIVars.g_maxGripAngle,		0,
	180,	-90-90,	60,				-90,											0,
	180,	-90-90,	60,				GVL_InstruTestUIVars.g_maxGripAngle,		0,
	0,		0-90,		0,				0,												0
	];
	m_GraspingForcepsTest: ARRAY [1..60, 1..5] OF LREAL:=
	[0,		0-90,		0,				0,		                                    0,	
	0,		0-90,		0,	     		GVL_InstruTestUIVars.g_maxGripAngle,		0,	
	0,		0-90,		0,				0,		 									0,	
	0,		0-90,		-60,			0,											0,	
	0,		0-90,		60,				0,											0,	
	0,		0-90,		0,				0,											0,
	0,		-60-90,	0,				0,											0,
	0,		60-90,		0,				0,											0,
	0,		0-90,		0,				0,											0,	
	180,	0-90,		0,				0,											0,	
	180,	0-90,		0,				GVL_InstruTestUIVars.g_maxGripAngle,		0,
	180,	0-90,		0,				0,											0,	
	180,	0-90,		-60,			0,											0,	
	180,	0-90,		60,			    0,											0,	
	180,	0-90,		0,				0,											0,	
	180,	-60-90,	0,				0,											0,	
	180,	60-90,		0,				0,											0,	
	  0,	0-90,		0,				0,											0,	
	-180,	0-90,		0,				0,											0,	 
	-180,	0-90,		0,				GVL_InstruTestUIVars.g_maxGripAngle,		0,	   
	-180,	0-90,		0,				0,											0,	 
	-180,	0-90,		-60,			0,											0,	   
	-180,	0-90,		60,				0,											0,	
	-180,	0-90,		0,				0,											0,	 
    -180,	-60-90,	0,				0,											0,	 
	-180,	60-90,		0,				0,											0,
	0,		0-90,		0,				0,											0,
	0,		0-90,		0,				0,											0
	];
	m_holdTheNeedleTest: ARRAY [1..60, 1..5] OF LREAL:=
	[0,		0-90,		0,				0,		                                        0,	
	0,		0-90,		0,	     		GVL_InstruTestUIVars.g_maxGripAngle,			0,	
	0,		0-90,		0,				-60,		 									0,	
	0,		0-90,		-60,			-60,											0,	
	0,		0-90,		60,				-60,											0,
	0,		0-90,		0,				-60,		 									0,	
	0,		-60-90,	0,				-60,		 									0,	
	0,		60-90,		0,				-60,		 									0,
	0,		0-90,		0,				-60,		 									0,
	180,	0-90,		0,				-60,		 									0,
	180,	0-90,		-60,			-60,		 									0,
	180,	0-90,		60,				-60,		 									0,
	180,	0-90,		0,				-60,		 									0,
	180,	-60-90,	0,				-60,		 									0,
	180,	60-90,		0,				-60,		 									0,
	180,	0-90,		0,				-60,		 									0,
	-180,	0-90,		0,				-60,		 									0,
	-180,	0-90,		-60,			-60,		 									0,
	-180,	0-90,		60,				-60,		 									0,
	-180,	0-90,		0,				-60,		 									0,
	-180,	-60-90,	0,				-60,		 									0,
	-180,	60-90,		0,				-60,		 									0,
	-180,	0-90,		0,				-60,		 									0,
	0,		0-90,		0,				0,		 										0,
	0,		0-90,		0,				0,		 										0
	];
	m_postureTest: ARRAY [1..60, 1..5] OF LREAL:=
	[0,		60-90,		0,				0,		0,	
	0,		-60-90,	0,	     		0,		0,	
	0,		0-90,		0,				0,	    0,	
	0,		0-90,		60,				0,	    0,
	0,		0-90,		-60,			0,	    0,
	0,		0-90,		0,				0,	    0,
	180,	0-90,		0,				0,	    0,
	0,		0-90,		0,				0,	    0,
	0,		0-90,		0,				GVL_InstruTestUIVars.g_maxGripAngle,	    0,
	0,		0-90,		0,				0,	    0,
	0,		0-90,		0,				GVL_InstruTestUIVars.g_minGripAngle,	    100,
	0,		0-90,		0,				0,	    0,
	0,		0-90,		0,				0,	    0,
	0,		0-90,		0,				0,	    0
	];
END_VAR

METHOD PROTECTED calcCmdJntPos : BOOL
VAR_IN_OUT CONSTANT
	i_endoscopePose : ST_Frame;
	i_masterStatus :ST_MasterStatus;
	i_setupStatus: ST_SetupStatus;
	i_slaveArm :FB_SlaveArm;
END_VAR

VAR 
	i:INT :=0;

